SettingsGetStr(
		sNetId:='',
		hFile:=hSettingsFile,
		bExecute:=bSettingsGetStrExecute,
		tTimeout:=T#1S,
		bBusy=>bSettingsGetStrBusy,
		bError=>bSettingsGetStrError,
		nErrId=>nSettingsGetStrError,
		sLine=>sSettingsGetStr,
		bEOF=>bGetStrSettingsEOF
);
		
SettingsClose(
		sNetId:='',
		hFile:=hSettingsFile,
		bExecute:=bSettingsCloseExecute,
		tTimeout:=T#5S,
		bBusy=>bSettingsCloseBusy,
		bError=>bSettingsCloseError,
		nErrId=>nSettingsCloseError
		);

END_PROGRAM

// ---- POUs/GENERAL/Components/Robot/ROBOTREMOTE.TcPOU
PROGRAM ROBOTREMOTE
VAR_INPUT
	bRobotCommOpenEnable : BOOL := FALSE;
	bRobotCommCloseEnable: BOOL := FALSE;
	bRobotCommandSend : BOOL := FALSE;
	sRobotCommand : STRING := '';
	sRobotCommandParam1 : STRING := '';
	sRobotCommandParam2 : STRING := '';
	sRobotCommandParam3 : STRING := '';
	sRobotCommandParam4 : STRING := '';
	sRobotCommandParam5 : STRING := '';
END_VAR
VAR_OUTPUT
	bRobotCommOpen : BOOL := FALSE;
	nRobotErrId: UDINT;
	sRobotResult : STRING := '';
	iState: INT := 0;
END_VAR
VAR	
//LOCALS
	//RobotComm
	sRobotRemoteHost: STRING := '192.168.1.100';
//	sRobotRemoteHost: STRING := '192.168.1.22';
	bConnectBusy: BOOL;
	bSendBusy: BOOL;
	bReceiveBusy: BOOL;
	bCloseBusy: BOOL;
	bConnectError: BOOL;
	bSendError: BOOL;
	bReceiveError: BOOL;
	bCloseError: BOOL;
	nConnectErrId: UDINT;
	nSendErrId: UDINT;
	nReceiveErrId: UDINT;
	nCloseErrId: UDINT;
	hRobotSocket: T_HSOCKET;
	Delay: TON;
	bStartDelay: BOOL := FALSE;
	tDelay: TIME;
	rDelay: REAL;
	bDelayTimePassed: BOOL;
	
	//Kapcsolat nyitás
	bRobotSocketOpenEnable: BOOL := FALSE;
	RobotSocketOpen: FB_SocketConnect;
	iOpenTrials: INT;
	
	//Küldés
	bExecuting : BOOL := FALSE;
	bRobotSocketSendEnable: BOOL := FALSE;
	RobotSocketSend: FB_SocketSend;
	sLRobotCommandForResult: STRING :='';
	sLRobotCommand: STRING :='';
	sLRobotParam1: STRING :='';
	sLRobotParam2: STRING :='';
	sLRobotParam3: STRING :='';
	sLRobotParam4: STRING :='';
	sLRobotParam5: STRING :='';
	sRobotSendData: STRING;
	uSendByteLen: UDINT := 0;
	baSendByteArray: ARRAY[0..255] OF BYTE;
	bRobotSocketReceiveEnable: BOOL := FALSE;
	RobotSocketReceive: FB_SocketReceive;
	sRobotReceived: STRING :='';
	nRobotReceivedBytesNum: UDINT;
	baReceivedByteArray: ARRAY[0..255] OF BYTE;
	iTemp : INT := 0;
	
	//Fogadás kiértékelés
	fb_ResultSplitter : fb_SplitRobotResult;
	bIsError : BOOL;
	sErrorOrResult : STRING;
	
	//Kapcsolat bontás
	bRobotSocketCloseEnable: BOOL := FALSE;
	RobotSocketClose: FB_SocketClose;
	bRobotSocketbusy: BOOL;
END_VAR

rDelay:=TIME_TO_REAL(tDelay);

RobotSocketOpen(
			sSrvNetId:= '', 
			sRemoteHost:= sRobotRemoteHost, 
			nRemotePort:= 5000, 
			bExecute:= bRobotSocketOpenEnable, 
			tTimeout:= T#90S, 
			bBusy=> bConnectBusy, 
			bError=> bConnectError, 
			nErrId=> nConnectErrId, 
			hSocket=> hRobotSocket);
			
RobotSocketSend(
		sSrvNetId:= '', 
		hSocket:= hRobotSocket, 
		cbLen:= uSendByteLen, 
		pSrc:= ADR(baSendByteArray), 
		bExecute:= bRobotSocketSendEnable, 
		tTimeout:= T#5S, 
		bBusy=> bSendBusy, 
		bError=> bSendError, 
		nErrId=> nSendErrId);
		
RobotSocketReceive(
	sSrvNetId:= '', 
	hSocket:= hRobotSocket, 
	cbLen:= 255, 
	pDest:= ADR(baReceivedByteArray), 
	bExecute:= bRobotSocketReceiveEnable, 
	tTimeout:= T#5S, 
	bBusy=> bReceiveBusy, 
	bError=> bReceiveError, 
	nErrId=> nReceiveErrId, 
	nRecBytes=> nRobotReceivedBytesNum);		
		
RobotSocketClose(
	sSrvNetId:= '', 
	hSocket:= hRobotSocket, 
	bExecute:= bRobotSocketCloseEnable, 
	tTimeout:= T#90S, 
	bBusy=> bCloseBusy, 
	bError=> bCloseError, 
	nErrId=> nCloseErrId);

//Kommunikáció nyitás
IF (bRobotCommOpenEnable = TRUE) AND (bRobotCommOpen = FALSE) AND (iState <= 0) THEN
	iState:=1;
	iOpenTrials:=0;
	bIsError:=FALSE;
END_IF;

//Parancs küldés
IF (bRobotCommandSend = TRUE) AND (bRobotCommOpen=TRUE) AND(iState <= 0) THEN
	iState:=11;
	bIsError:=FALSE;
END_IF;
//Kommunikáció zárás
IF (bRobotCommCloseEnable = TRUE) AND (bRobotCommOpen = TRUE) AND (iState <= 0) THEN
	iState:=31;
	bIsError:=FALSE;
END_IF;




CASE iState OF
	
	1:	//Kommunikáció nyitás
		bRobotSocketOpenEnable:=TRUE;
		iState:=2;
	
	2:
		IF bConnectBusy = TRUE THEN
			iState:=3;
		END_IF
	3:
		IF bConnectBusy = FALSE THEN
			iState:=4;
		END_IF 
		
	4:
		IF bConnectError =FALSE THEN
			//Minden OK
			bRobotCommOpen:=TRUE;
			iState:=0;
		ELSE
			//HIBA
			iOpenTrials:=iOpenTrials+1;
			bRobotCommOpen:=FALSE;
			IF iOpenTrials<6 THEN
				bConnectError:=FALSE;
				iState:=5;
				bStartDelay:=TRUE;
				tDelay:=T#10S;
			ELSE
				iOpenTrials:=0;
				bStartDelay:=FALSE;
				iState:=0;
			END_IF
		END_IF
		bRobotCommOpenEnable := FALSE;
		bRobotSocketOpenEnable:=FALSE;
	5:
		IF bDelayTimePassed=TRUE THEN
			bStartDelay:=FALSE;
			iState:=1;
		END_IF
		
		
	11: //Parancs küldés
		nRobotErrId := 0;
		sLRobotCommandForResult := sRobotCommand;
		sLRobotCommand := sRobotCommand;
		sLRobotParam1 := sRobotCommandParam1;
		sLRobotParam2 := sRobotCommandParam2;
		sLRobotParam3 := sRobotCommandParam3;
		sLRobotParam4 := sRobotCommandParam4;
		sLRobotParam5 := sRobotCommandParam5;
		sRobotSendData := f_RobotCommandTranslation(sLRobotCommand,sLRobotParam1,sLRobotParam2,sLRobotParam3,sLRobotParam4,sLRobotParam5);
		baSendByteArray := MAXSTRING_TO_BYTEARR(sRobotSendData);
		uSendByteLen := INT_TO_UDINT(LEN(sRobotSendData));
		MEMSET(ADR(baReceivedByteArray), 0, 256);
		
		iState:=12;
		
	12:
		bRobotSocketSendEnable:=TRUE;
		iState:=13;
		
	13:
		IF bSendBusy = TRUE THEN
			iState:=14;
		END_IF
	14:
		IF bSendBusy = FALSE THEN
			iState:=15;
		END_IF 
		
	15:
		IF bSendError =FALSE THEN
			//Minden OK
			bIsError:= FALSE;
			iState:=21;
		ELSE
			//HIBA
			bIsError:= TRUE;	
			iState:=0;
		END_IF
		bRobotCommandSend := FALSE;
		bRobotSocketSendEnable:=FALSE;
		
		sRobotCommand:='';
		sRobotCommandParam1 := '';
		sRobotCommandParam2 := '';
		sRobotCommandParam3 := '';
		sRobotCommandParam4 := '';
		sRobotCommandParam5 := '';
		
		sLRobotCommand := '';
		sLRobotParam1 := '';
		sLRobotParam2 := '';
		sLRobotParam3 := '';
		sLRobotParam4 := '';
		sLRobotParam5 := '';
		
	21:	//Adatfogadás
		nRobotReceivedBytesNum:=0;
		bRobotSocketReceiveEnable := TRUE;
		iState:=22;
		
	22:
		IF bReceiveBusy = TRUE THEN
			iState:=23;
		END_IF
	23:
		IF bReceiveBusy = FALSE THEN
			iState:=24;
		END_IF 
		
	24:
		IF bReceiveError =FALSE THEN
			//Minden OK
			bIsError:= FALSE;
			iState:=25;
		ELSE
			//HIBA
			bIsError:= TRUE;
			iState:=0;	
		END_IF
		bRobotSocketReceiveEnable:=FALSE;
		
	25:
		IF (nRobotReceivedBytesNum <>0) THEN
			sRobotReceived := BYTEARR_TO_MAXSTRING(baReceivedByteArray);
			fb_ResultSplitter(sCommand:= sLRobotCommandForResult, sResult:= sRobotReceived, bIsError=> bIsError, sErrorOrResult=> sErrorOrResult);
			IF bIsError THEN
				nRobotErrId:=STRING_TO_UDINT(sErrorOrResult);
				sRobotResult:='';
			ELSE
				nRobotErrId:=0;
				sRobotResult:=sErrorOrResult;
			END_IF
			iState:=0;
		ELSE
			iState:=21;
		END_IF
		
	31:	//Kommunikáció zárás
		bRobotSocketCloseEnable:=TRUE;
		iState:=32;
	
	32:
		IF bCloseBusy = TRUE THEN
			iState:=33;
		END_IF
	33:
		IF bCloseBusy = FALSE THEN
			iState:=34;
		END_IF 
		
	34:
		IF bCloseError =FALSE THEN
			//Minden OK
			bRobotCommOpen:=FALSE;
		ELSE
			//HIBA
			bRobotCommOpen:=FALSE;	//még át kell gondolni
		END_IF
		bRobotCommCloseEnable := FALSE;
		bRobotSocketCloseEnable:=FALSE;
		iState:=0;
	
END_CASE
Delay(IN:=bStartDelay, PT:=tDelay, Q=>bDelayTimePassed, ET=>);

END_PROGRAM

// ---- POUs/GENERAL/Helpers/fb_SplitRobotResult.TcPOU
FUNCTION_BLOCK fb_SplitRobotResult
VAR_INPUT
	sCommand : STRING;
	sResult : STRING;
END_VAR
VAR_OUTPUT
	bIsError : BOOL;
	sErrorOrResult : STRING;
END_VAR
VAR
	sCRLFString : STRING := '  ';
	nCRLFPosition : INT := 0;
	sTempResult : STRING;
END_VAR

sCRLFString[0] := 16#D;
sCRLFString[1] := 16#A;
IF MID(sResult,LEN(sCommand),2)=sCommand THEN
	sErrorOrResult := MID(sResult,LEN(sResult)-LEN(sCommand)-4,3+LEN(sCommand));
	nCRLFPosition := FIND(sErrorOrResult,sCRLFString);
	IF nCRLFPosition > 0 THEN
		sErrorOrResult := DELETE(sErrorOrResult,2,nCRLFPosition);
	END_IF
	IF sResult[0] = 16#23 THEN
		bIsError := FALSE;
	ELSE
		bIsError := TRUE;
	END_IF
ELSE
	bIsError := TRUE;
	sErrorOrResult := '1';
END_IF

END_FUNCTION_BLOCK

// ---- POUs/GENERAL/Helpers/f_RobotCommandTranslation.TcPOU
FUNCTION f_RobotCommandTranslation : STRING
VAR_INPUT
	sCommand : STRING;
	sParam1 : STRING;
	sParam2 : STRING;
	sParam3 : STRING;
	sParam4 : STRING;
	sParam5 : STRING;
END_VAR
VAR
	uLength : INT := 0;
	tempTranslation : STRING := '';
	nDollarPosition : INT := 0;
	sDollarString : STRING := ' ';
END_VAR

//IF sCommand='Login' THEN
//	f_RobotCommandTranslation := CONCAT(' Login,',sParam1);
//END_IF
//IF sCommand='LOGOUT' THEN
//	f_RobotCommandTranslation:=' Logout';
//END_IF
//Kezdő $ karakter
sDollarString[0] := 16#24;
tempTranslation := CONCAT(' ',sCommand);
tempTranslation[0] := 16#24;

//Ha van Paraméter1 akkor berakjuk
IF sParam1<>'' THEN
	tempTranslation := CONCAT(tempTranslation,',');
	tempTranslation := CONCAT(tempTranslation,sParam1);
END_IF

//Ha van Paraméter2 akkor berakjuk
IF sParam2<>'' THEN
	tempTranslation := CONCAT(tempTranslation,',');
	tempTranslation := CONCAT(tempTranslation,sParam2);
END_IF

//Ha van Paraméter3 akkor berakjuk
IF sParam3<>'' THEN
	tempTranslation := CONCAT(tempTranslation,',');
	tempTranslation := CONCAT(tempTranslation,sParam3);
END_IF

//Ha van Paraméter4 akkor berakjuk
IF sParam4<>'' THEN
	tempTranslation := CONCAT(tempTranslation,',');
	tempTranslation := CONCAT(tempTranslation,sParam4);
END_IF

//Ha van Paraméter5 akkor berakjuk
IF sParam5<>'' THEN
	tempTranslation := CONCAT(tempTranslation,',');
	tempTranslation := CONCAT(tempTranslation,sParam5);
END_IF

//Add CRLF to end
tempTranslation := CONCAT(tempTranslation,'  ');
tempTranslation[LEN(tempTranslation)-2]:=16#D;
tempTranslation[LEN(tempTranslation)-1]:=16#A;
nDollarPosition := FIND(tempTranslation,'dollar');
IF nDollarPosition > 0 THEN
	tempTranslation := DELETE(tempTranslation,6,nDollarPosition);
	tempTranslation := INSERT(tempTranslation,sDollarString,nDollarPosition-1);
END_IF
f_RobotCommandTranslation:=tempTranslation;

END_FUNCTION

// ---- POUs/PISTI/Components/Laser.TcPOU
PROGRAM Laser
VAR_INPUT
	s_InCommand : STRING :='';
	s_TypeCode : STRING :='0';	
END_VAR
VAR_OUTPUT
	s_Result: STRING;
END_VAR
VAR
	iState: INT;
	iState2: INT;
	iTrials: INT;
	iSetPower: INT;
	iWishPower: INT := 12;
	sWishPower: STRING;
	sSetPower: STRING;

	// Laser Com Open
	sLaserRemoteHost: STRING := '192.168.1.99';
//	sLaserRemoteHost: STRING := '192.168.1.22';
	LaserSocketOpen: FB_SocketConnect;
	bLaserSocketOpenEnable: BOOL := FALSE;
	bLaserSocketBusy: BOOL;
	bLaserSocketError: BOOL;
	nLaserSocketErrId: UDINT;
	hLaserSocket: T_HSOCKET;
	
	// Laser Send
	LaserSocketSend: FB_SocketSend;
	uSendByteLen: UDINT := 0;
	baSendByteArray: ARRAY[0..255] OF BYTE;
	bLaserSocketSendEnable: BOOL := FALSE;
	bLaserSendbusy: BOOL;
	bLaserSendError: BOOL;
	nLaserSendErrId: UDINT;

	// Laser Receive
	LaserSocketReceive: FB_SocketReceive;
	baReceivedByteArray: ARRAY[0..255] OF BYTE;
	bLaserSocketReceiveEnable: BOOL := FALSE;
	bLaserReceiveBusy: BOOL;
	bLaserReceiveError: BOOL;
	nLaserReceiveErrId: UDINT;
	nLaserReceivedBytesNum: UDINT;
	
	// Laser Com Close
	LaserSocketClose: FB_SocketClose;
	bLaserSocketCloseEnable: BOOL := FALSE;
	bLaserSocketCloseBusy: BOOL;
	bLaserSocketCloseError: BOOL;
	nLaserSocketCloseErrId: UDINT;
	
	sLaserSend: STRING :='';
	sLaserReceived: STRING :='';
	sExpectedResponse: STRING := '';
	
	// Lézer szoftver megnyitása
	FB_Start_FOBA_Draw: NT_StartProcess;
	bStartFOBADraw: BOOL;
	bFOBADrawBusy: BOOL;
	bFOBADrawErr: BOOL;
	nFOBADrawErr: UDINT;

	// Lézer parancs lista megnyitása
	FB_Start_Ultimate: NT_StartProcess;
	bStartUltimate: BOOL;
	bUltimateBusy: BOOL;
	bUltimateErr: BOOL;
	nUltimateErr: UDINT;
	
END_VAR

CASE iState OF
	0:	// Parancsértelmezés
		iState:=1;
		iTrials:=0;
		sExpectedResponse:='$06;0000;$R$N';
		IF s_InCommand='GETJOB' THEN
			sLaserSend:='GetJob;';
		ELSIF s_InCommand='SETJOB_637' THEN
			sLaserSend:='SetJob;637xxx;';
		ELSIF s_InCommand='SETJOB_745900' THEN
			sLaserSend:='SetJob;745900;';
		ELSIF s_InCommand='SETJOB_745910' THEN
			sLaserSend:='SetJob;745910;';
		ELSIF s_InCommand='SETJOB_521' THEN
			sLaserSend:='SetJob;521950;';
		ELSIF s_InCommand='START' THEN
			sLaserSend:='Start;';
		ELSIF (s_InCommand='SETTYPE') THEN
			IF (GVL.iSelectedProductType<8) THEN // 637 esetén
				s_TypeCode:=TO_STRING(GVL.iSelectedProductType);
			ELSIF (GVL.iSelectedProductType>8) THEN // 745 esetén
				CASE GVL.iSelectedProductType OF
					9, 10: s_TypeCode:='0'; //745900 és 745910
					11, 12: s_TypeCode:='1'; //745905 és 745915
					13, 14: s_TypeCode:='2'; //745906 és 745916
					15, 16: s_TypeCode:='3'; //745907 és 745917
				END_CASE
			END_IF;
			sLaserSend:=CONCAT('SetVars;TypeCode;',CONCAT(s_TypeCode,';'));
		ELSIF s_InCommand='GETSTATUS' THEN
			sLaserSend:='GetStatus;';
			s_Result:='';
		ELSIF s_InCommand='GETINTENSITY' THEN
			sLaserSend:='GetIntensity;';
			s_Result:='';
		ELSE
			iState:=0;
		END_IF			
	1:	// Vár arra, hogy ne legyen folyamatban a socket megnyitása
		IF (bLaserSocketBusy=FALSE) THEN
			iState:=2;
		END_IF							
	2:	// Ha nincs nyitva a lézer socket, kezdeményezi a megnyitását
		IF NOT(GVL.bLaserCommOpen) THEN
			bLaserSocketOpenEnable:=TRUE;
			IF (bLaserSocketBusy=TRUE) THEN
				iState:=3;
			END_IF				
		ELSE
			iState:=4;
		END_IF
	3:	// Vár, hogy megnyíljon a lézer socket
		IF (bLaserSocketBusy=FALSE) AND (bLaserSocketError=FALSE) THEN
			GVL.bLaserCommOpen:=TRUE;
			bLaserSocketOpenEnable:=FALSE;
			iState:=4;
		ELSIF (bLaserSocketError=TRUE) THEN
			GVL.bLaserCommOpen:=FALSE;
			bLaserSocketOpenEnable:=FALSE;
			iState:=2;
		END_IF
	4:	// Ha nincs folyamatban parancsküldés, kezdeményezi a parancsküldést
		IF (bLaserSendBusy=FALSE) THEN
			MEMSET(ADR(baSendByteArray), 0, 256); // Byte tömb ürítése
			baSendByteArray := MAXSTRING_TO_BYTEARR(sLaserSend); // Parancs string byte tömbbe
			uSendByteLen := INT_TO_UDINT(LEN(sLaserSend)); // Parancs string hossza
			baSendByteArray[uSendByteLen]:=16#D; // Lezáró karakter 1
			baSendByteArray[uSendByteLen+1]:=16#A; // Lezáró karakter 2
			bLaserSocketSendEnable:=TRUE; // Küldés indítójel
			iState:=5;
		END_IF
	5:	// Vár, hogy a parancsküldés elkezdődjön
		IF (bLaserSendBusy=TRUE) THEN
			iState:=6;
		END_IF
	6:	// Vár a parancsküldés sikeres befejezésére
		IF (bLaserSendBusy=FALSE) AND (bLaserSendError=FALSE) THEN
			bLaserSocketSendEnable:=FALSE;
			iState:=7;
		END_IF
	7:	// Ha nincs folyamatban válaszfogadás, kezdeményezi a válaszfogadást
		IF (bLaserReceiveBusy=FALSE) THEN
			MEMSET(ADR(baReceivedByteArray), 0, 256); // Byte tömb ürítése
			bLaserSocketReceiveEnable:=TRUE; // Fogadás indítójel
			iState:=8;
		END_IF
	8:	// Vár, hogy a válaszfogadás elkezdődjön
		IF (bLaserReceiveBusy=TRUE) THEN
			iState:=9;
		END_IF
	9:	// Vár a válaszfogadás sikeres befejezésére
		IF (bLaserReceiveBusy=FALSE) AND (bLaserReceiveError=FALSE) THEN
			bLaserSocketReceiveEnable:=FALSE;
			sLaserReceived := BYTEARR_TO_MAXSTRING(baReceivedByteArray);
			MEMSET(ADR(baReceivedByteArray), 0, 256);
			iState:=10;
		END_IF
	10:	// Kiértékelés
		IF (sLaserReceived=sExpectedResponse) THEN
			s_InCommand:='';
		ELSE
			IF iTrials<5 THEN
				iTrials:=iTrials+1;
				iState:=7;
			ELSE
				s_InCommand:=sLaserReceived;
			END_IF
		END_IF
		sExpectedResponse:='';
		iState:=0;
		IF sLaserSend='GetStatus;' THEN
			IF (FIND(sLaserReceived,'LaserStatusReady')>0)
				OR (FIND(sLaserReceived,'LaserStatusStandby')>0) THEN
				s_Result:='READY';
			ELSE
				s_Result:='NOT_READY';
			END_IF
		ELSIF LEFT(sLaserSend,12)='GetIntensity' THEN
			sSetPower:=DELETE(sLaserReceived,8,0);
			sSetPower:=LEFT(sSetPower,LEN(sSetPower)-3);
			iSetPower:=STRING_TO_INT(sSetPower);
//			sLaserSend:='GetIntensity;';
			;
		ELSIF LEFT(sLaserSend,12)='SetIntensity' THEN
			sLaserSend:='GetIntensity;';
			iState:=1;
		END_IF
END_CASE

// FOBA Draw indítási állapotgép
CASE iState2 OF
	0:	// Várakozás parancsra
		IF (bStartFOBADraw=TRUE) THEN
			iState2:=1;
		ELSIF (bStartUltimate=TRUE) THEN
			iState2:=11;
		END_IF
	1:
		IF (bFOBADrawBusy=TRUE) THEN
			iState2:=2;
		END_IF
	2:
		IF (bFOBADrawBusy=FALSE) THEN
			bStartFOBADraw:=FALSE;
			iState2:=0;
		END_IF
	11:
		IF (bUltimateBusy=TRUE) THEN
			iState2:=12;
		END_IF
	12:
		IF (bUltimateBusy=FALSE) THEN
			bStartUltimate:=FALSE;
			iState2:=0;
		END_IF
END_CASE

// Kommunikáció nyitás
LaserSocketOpen(
	sSrvNetId:= '', 
	sRemoteHost:= sLaserRemoteHost, 
	nRemotePort:= 20001, 
	bExecute:= bLaserSocketOpenEnable, 
	tTimeout:= T#45S, 
	bBusy=> bLaserSocketBusy, 
	bError=> bLaserSocketError, 
	nErrId=> nLaserSocketErrId, 
	hSocket=> hLaserSocket);

// Parancsküldés
LaserSocketSend(
	sSrvNetId:= '', 
	hSocket:= hLaserSocket, 
	cbLen:= uSendByteLen + 2, 
	pSrc:= ADR(baSendByteArray), 
	bExecute:= bLaserSocketSendEnable, 
	tTimeout:= T#5S, 
	bBusy=> bLaserSendBusy,
	bError=> bLaserSendError,
	nErrId=> nLaserSendErrId);

// Válasz fogadása
LaserSocketReceive(
	sSrvNetId:= '', 
	hSocket:= hLaserSocket, 
	cbLen:= 255, 
	pDest:= ADR(baReceivedByteArray), 
	bExecute:= bLaserSocketReceiveEnable, 
	tTimeout:= T#5S, 
	bBusy=> bLaserReceiveBusy, 
	bError=> bLaserReceiveError, 
	nErrId=> nLaserReceiveErrId, 
	nRecBytes=> nLaserReceivedBytesNum
);

//Kommunikáció bontás
LaserSocketClose(
	sSrvNetId:= '', 
	hSocket:= hLaserSocket, 
	bExecute:= bLaserSocketCloseEnable, 
	tTimeout:= T#45S, 
	bBusy=> bLaserSocketCloseBusy, 
	bError=> bLaserSocketCloseError, 
	nErrId=> nLaserSocketCloseErrId);

// Lézer saját szoftverének indítása
FB_Start_FOBA_Draw(
					NETID:='',
					PATHSTR:='C:\Program Files\FOBA\FOBA Draw\FOBA Draw 9.2.2\FOBA Draw.exe',
					DIRNAME:='C:\Program Files\FOBA\FOBA Draw\FOBA Draw 9.2.2\',
					COMNDLINE:='',
					START:=bStartFOBADraw,
					TMOUT:=T#30S,
					BUSY => bFOBADrawBusy,
					ERR => bFOBADrawErr,
					ERRID => nFOBADrawErr
					);

// Lézer parancs listájának megnyitása
FB_Start_Ultimate(
					NETID:='',
					PATHSTR:='C:\Program Files\Adobe\Reader 11.0\Reader\AcroRd32.exe',
					DIRNAME:='C:\637\',
					COMNDLINE:='"C:\637\Specification_Ultimate_V1.5.1_Foba_Rev2.pdf"',
					START:=bStartUltimate,
					TMOUT:=T#30S,
					BUSY => bUltimateBusy,
					ERR => bUltimateErr,
					ERRID => nUltimateErr
					);

END_PROGRAM

// ---- POUs/JOZSI/Components/NTC.TcPOU
PROGRAM NTC
VAR_INPUT
	bVagashoz : BOOL := FALSE;

	//Gombok funkcióváltása
	bVagasGombbal : BOOL;
	bVagoFelLeGombbal : BOOL;
END_VAR
VAR
	
	//IO
	bZoldGomb AT %I*: BOOL;
	bPirosGomb AT %I*: BOOL;
	bNTCLaberzekeloBal AT %I*: BOOL;
	bNTCLaberzekeloJobb AT %I*: BOOL;
	bNTCFekBal AT %Q*: BOOL := FALSE;
	bNTCFekJobb AT %Q*: BOOL := FALSE;
	
	
	//MOTOR
	bZeroSpeed AT %I*: BOOL;
	bSpeedReached AT %I*: BOOL;
	bReady AT %I*: BOOL;
	bAlarm AT %I*: BOOL;
	bServoON AT %Q*: BOOL := TRUE;
	bReverseRotationStart AT %Q*: BOOL := FALSE;
	bForwardRotationStart AT %Q*: BOOL := FALSE;
	bSpeed1 AT %Q*: BOOL := TRUE;
	bReset AT %Q*: BOOL := FALSE;
	
	//VARS
	bInternalState : BOOL := FALSE;
	iDelayFor : INT := 0;
	iTemp : INT := 0;
	bJogPlus : BOOL := FALSE;
	bJogMinus : BOOL := FALSE;
	bElozoLab : BOOL := FALSE;
	
	
END_VAR

IF (bVagasGombbal=FALSE) AND (bVagoFelLeGombbal=FALSE) THEN
	IF ((bZoldGomb=TRUE OR bJogPlus=TRUE) AND bAlarm=TRUE AND bServoON=TRUE AND bReady=TRUE) THEN
		bForwardRotationStart := TRUE;
		bReverseRotationStart := FALSE;
		bVagashoz:=FALSE;
		bInternalState:=FALSE;
	ELSE
		IF bInternalState=FALSE THEN
			bForwardRotationStart := FALSE;
		END_IF
	END_IF
	IF ((bPirosGomb=TRUE OR bJogMinus=TRUE) AND bAlarm=TRUE AND bServoON=TRUE AND bReady=TRUE) THEN
		bReverseRotationStart := TRUE;
		bForwardRotationStart := FALSE;
		bVagashoz:=FALSE;
		bInternalState:=FALSE;
	ELSE
		IF bInternalState=FALSE THEN
			bReverseRotationStart := FALSE;
		END_IF
	END_IF
ELSIF (bVagoFelLeGombbal=TRUE) AND (NTCProcess.s_InCommand='')
		AND ((bZoldGomb=TRUE) OR (bPirosGomb=TRUE)) THEN
	NTCProcess.s_InCommand:='VAGO_FEL-LE';
ELSIF (bZoldGomb=TRUE) AND (NTCProcess.s_InCommand='') THEN
	NTCProcess.s_InCommand:='VAGAS';
ELSIF (bPirosGomb=TRUE) AND (NTCProcess.s_InCommand='') THEN
	NTCProcess.s_InCommand:='NTC_ELENGED';
END_IF;

(*// Új NTC pozícionáló algoritmus (két lábérzékelő + két fék)	
IF (bVagashoz=TRUE AND bAlarm=TRUE AND bServoON=TRUE AND bReady=TRUE) THEN
	bInternalState := TRUE;
	bVagashoz:=FALSE;
	IF (bNTCLaberzekeloBal=TRUE) AND (bNTCLaberzekeloJobb=TRUE) THEN
		bElozoLab := TRUE;
	END_IF
END_IF
		
IF bInternalState=TRUE THEN
//	IF (bNTCLaberzekeloBal=TRUE) AND (bNTCLaberzekeloJobb=TRUE) THEN		
	IF (bNTCFekBal=TRUE) AND (bNTCFekJobb=TRUE) THEN		
		bNTCFekBal:=FALSE;
		bNTCFekJobb:=FALSE;
		IF bElozoLab=FALSE THEN
			bForwardRotationStart := FALSE;
			bInternalState := FALSE;
		ELSE
			bForwardRotationStart := TRUE;
		END_IF
	ELSIF (bNTCLaberzekeloBal=TRUE) THEN
		bNTCFekBal:=TRUE;
	ELSIF (bNTCLaberzekeloJobb=TRUE) THEN
		bNTCFekJobb:=TRUE;
	ELSE	
		IF bElozoLab = TRUE THEN
			bElozoLab := FALSE;
		END_IF;
		bForwardRotationStart := TRUE;
	END_IF
END_IF
*)
// Régi NTC pozícionáló algoritmus: csak egy lábérzékelő fékek nélkül
IF (bVagashoz=TRUE AND bAlarm=TRUE AND bServoON=TRUE AND bReady=TRUE) THEN
	bInternalState := TRUE;
	bVagashoz:=FALSE;
	IF(bNTCLaberzekeloJobb=TRUE) THEN
		bElozoLab := TRUE;
	END_IF
END_IF
		
IF bInternalState=TRUE THEN
	IF(bNTCLaberzekeloJobb=TRUE) THEN
		IF bElozoLab=FALSE THEN
			bForwardRotationStart := FALSE;
			bInternalState := FALSE;
		ELSE
			bForwardRotationStart := TRUE;
		END_IF
	ELSE
		IF bElozoLab = TRUE THEN
			bElozoLab := FALSE;
		END_IF;
		bForwardRotationStart := TRUE;
	END_IF
END_IF

END_PROGRAM

// ---- POUs/JOZSI/Components/NTCProcess.TcPOU
PROGRAM NTCProcess
VAR_INPUT
	s_InCommand : STRING := '';
	s_InCommandParam1 : STRING := '';
	s_InCommandParam2 : STRING := '';
	s_InCommandParam3 : STRING := '';
	s_InCommandParam4 : STRING := '';
	s_InCommandParam5 : STRING := '';
END_VAR
VAR_OUTPUT
	n_OutErrId: UINT;
END_VAR
VAR
	//IO
	bVagoHajlitoFent AT %I*: BOOL;
	bVagoHajlitoLent AT %I*: BOOL;
	bKiszedoKint AT %I*: BOOL;
	bKiszedoBent AT %I*: BOOL;
	bMegfogoNyitva AT %I*: BOOL;
	bMegfogoZarva AT %I*: BOOL;
	bVagoHajlito AT %Q*: BOOL := FALSE;
	bKiszedo AT %Q*: BOOL := FALSE;
	bMegfogo AT %Q*: BOOL := FALSE;
	
	//INTERNAL	
	iState : INT := 0;
	s_InLCommand : STRING := '';
	T_Ticker : TON;
	bTickerEnable : BOOL := FALSE;
	tTickerTime : TIME := T#3000MS;
	bTickerQ : BOOL := FALSE;
END_VAR

IF NTCProcess.s_InCommand <>'' AND s_InLCommand = '' THEN
	s_InLCommand := NTCProcess.s_InCommand;
END_IF
IF s_InLCommand <> '' THEN
//	IF iState = 0 AND s_InLCommand = 'VAGAS' THEN
//		iState := 1;
//	END_IF
	IF iState = 0 THEN 
		IF s_InLCommand = 'VAGAS' THEN
			iState := 1;
		ELSIF s_InLCommand = 'NTC_ELENGED' THEN
			iState := 21;
		ELSIF s_InLCommand = 'VAGO_FEL-LE' THEN
			iState := 31;
		END_IF
	END_IF
	CASE iState OF 
		1:
			IF (bVagoHajlitoFent = TRUE AND bVagoHajlitoLent = FALSE
				AND bKiszedoBent = FALSE AND bKiszedoKint = TRUE
				AND bMegfogoZarva = FALSE AND bMegfogoNyitva = TRUE
				AND NTC.bInternalState=FALSE) THEN
				n_OutErrId := 0;
				iState := 2;
			ELSE
				IF MAIN.bLevegoOK = FALSE THEN
					n_OutErrId := 5;
				ELSIF bVagoHajlitoFent = FALSE THEN
					n_OutErrId := 115;
				ELSIF bVagoHajlitoLent = TRUE THEN
					n_OutErrId := 114;
				ELSIF bKiszedoBent = TRUE THEN
					n_OutErrId := 136;
				ELSIF bKiszedoKint = FALSE THEN
					n_OutErrId := 133;
				ELSIF bMegfogoZarva = TRUE THEN 
					n_OutErrId := 132;
				ELSIF bMegfogoNyitva = FALSE THEN
					n_OutErrId := 129;
				ELSIF NTC.bInternalState=TRUE THEN
					n_OutErrId := 300;
				END_IF;
				iState := 0;
			END_IF
		2:
			NTC.bVagashoz := TRUE;
			iState := 3;
		3:
			IF (NTC.bInternalState = FALSE AND NTC.bVagashoz = FALSE) THEN
				iState := 4;
				n_OutErrId := 0;
			ELSIF NTC.bInternalState=TRUE THEN
				n_OutErrId := 300;
			ELSIF NTC.bVagashoz = TRUE THEN
				n_OutErrId := 301;
			END_IF
		4:
			bKiszedo := TRUE;
			iState := 5;
		5:
			IF bKiszedoBent = TRUE AND bKiszedoKint = FALSE THEN
				n_OutErrId := 0;
				tTickerTime:=T#1S;
				bTickerEnable := FALSE;
				iState := 6;
			ELSIF MAIN.bLevegoOK = FALSE THEN
				n_OutErrId := 5;
			ELSIF bKiszedoBent = FALSE THEN
				n_OutErrId := 135;
			ELSIF bKiszedoKint = TRUE THEN
				n_OutErrId := 134;
			END_IF
		6:
			bTickerEnable := TRUE;
			iState := 7;
		7:
			IF bTickerQ = TRUE THEN
				bTickerEnable := FALSE;
				iState := 8;
			END_IF
		8:
			bVagoHajlito := TRUE;
			iState := 9;
		9:
			IF bVagoHajlitoLent = TRUE AND bVagoHajlitoFent = FALSE THEN
				n_OutErrId := 0;
				tTickerTime:=T#1S;
				bTickerEnable := FALSE;
				iState := 10;
			ELSIF MAIN.bLevegoOK = FALSE THEN
				n_OutErrId := 5;
			ELSIF bVagoHajlitoLent = FALSE THEN 
				n_OutErrId := 113;
			ELSIF bVagoHajlitoFent = TRUE THEN
				n_OutErrId := 116;
			END_IF
		10:
			bTickerEnable := TRUE;
			iState := 11;
		11:
			IF bTickerQ = TRUE THEN
				bTickerEnable := FALSE;
				iState := 12;
			END_IF
		12:
			bVagoHajlito := FALSE;
			iState := 13;
		13:
			IF bVagoHajlitoLent = FALSE AND bVagoHajlitoFent = TRUE THEN
				n_OutErrId := 0;
				tTickerTime:=T#3S;
				bTickerEnable := FALSE;
				iState := 14;
			ELSIF MAIN.bLevegoOK = FALSE THEN
				n_OutErrId := 5;
			ELSIF bVagoHajlitoLent = TRUE THEN 
				n_OutErrId := 114;
			ELSIF bVagoHajlitoFent = FALSE THEN
				n_OutErrId := 115;
			END_IF
		14:
			bTickerEnable := TRUE;
			iState := 15;
		15:
			IF bTickerQ = TRUE THEN
				bTickerEnable := FALSE;
				iState := 16;
			END_IF
		16:
			bMegfogo := TRUE;
			iState := 17;
		17:
			IF bMegfogoZarva = TRUE AND bMegfogoNyitva = FALSE THEN
				n_OutErrId := 0;
				iState := 18;
			ELSIF MAIN.bLevegoOK = FALSE THEN
				n_OutErrId := 5;
			ELSIF bMegfogoZarva = FALSE THEN 
				n_OutErrId := 131;
			ELSIF bMegfogoNyitva = TRUE THEN
				n_OutErrId := 130;
			END_IF
		18:
			bKiszedo := FALSE;
			iState := 19;
		19:
			IF bKiszedoKint = TRUE AND bKiszedoBent = FALSE THEN
				n_OutErrId := 0;
				iState := 20;
			ELSIF MAIN.bLevegoOK = FALSE THEN
				n_OutErrId := 5;
			ELSIF bKiszedoKint = FALSE THEN 
				n_OutErrId := 133;
			ELSIF bKiszedoBent = TRUE THEN
				n_OutErrId := 136;
			END_IF
		20:
			iState := 0;
			n_OutErrId := 0;
		21:
			bMegfogo := FALSE;
			iState := 22;

		22:
			IF bMegfogoZarva = FALSE AND bMegfogoNyitva = TRUE THEN
				n_OutErrId := 0;
				iState := 20;
			ELSIF MAIN.bLevegoOK = FALSE THEN
				n_OutErrId := 5;
			ELSIF bMegfogoZarva = TRUE THEN 
				n_OutErrId := 132;
			ELSIF bMegfogoNyitva = FALSE THEN
				n_OutErrId := 129;
			END_IF

		31:
			IF (bVagoHajlitoFent = TRUE AND bVagoHajlitoLent = FALSE
				AND bKiszedoBent = FALSE AND bKiszedoKint = TRUE
				AND bMegfogoZarva = FALSE AND bMegfogoNyitva = TRUE
				AND NTC.bInternalState=FALSE) THEN
				n_OutErrId := 0;
				iState := 32;
			ELSE
				IF MAIN.bLevegoOK = FALSE THEN
					n_OutErrId := 5;
				ELSIF bVagoHajlitoFent = FALSE THEN
					n_OutErrId := 115;
				ELSIF bVagoHajlitoLent = TRUE THEN
					n_OutErrId := 114;
				ELSIF bKiszedoBent = TRUE THEN
					n_OutErrId := 136;
				ELSIF bKiszedoKint = FALSE THEN
					n_OutErrId := 133;
				ELSIF bMegfogoZarva = TRUE THEN 
					n_OutErrId := 132;
				ELSIF bMegfogoNyitva = FALSE THEN
					n_OutErrId := 129;
				ELSIF NTC.bInternalState=TRUE THEN
					n_OutErrId := 300;
				END_IF;
				iState := 0;
			END_IF
		32:
			bVagoHajlito := TRUE;
			iState := 33;
		33:
			IF bVagoHajlitoLent = TRUE AND bVagoHajlitoFent = FALSE THEN
				n_OutErrId := 0;
				tTickerTime:=T#1S;
				bTickerEnable := FALSE;
				iState := 34;
			ELSIF MAIN.bLevegoOK = FALSE THEN
				n_OutErrId := 5;
			ELSIF bVagoHajlitoLent = FALSE THEN 
				n_OutErrId := 113;
			ELSIF bVagoHajlitoFent = TRUE THEN
				n_OutErrId := 116;
			END_IF
		34:
			bTickerEnable := TRUE;
			iState := 35;
		35:
			IF bTickerQ = TRUE THEN
				bTickerEnable := FALSE;
				iState := 36;
			END_IF
		36:
			bVagoHajlito := FALSE;
			iState := 37;
		37:
			IF bVagoHajlitoLent = FALSE AND bVagoHajlitoFent = TRUE THEN
				n_OutErrId := 0;
				iState := 0;
			ELSIF MAIN.bLevegoOK = FALSE THEN
				n_OutErrId := 5;
			ELSIF bVagoHajlitoLent = TRUE THEN 
				n_OutErrId := 114;
			ELSIF bVagoHajlitoFent = FALSE THEN
				n_OutErrId := 115;
			END_IF

	END_CASE
	IF iState = 0 THEN
		NTCProcess.s_InCommand := '';
		s_InLCommand := '';
	END_IF
END_IF
T_Ticker(IN:= bTickerEnable, PT:= tTickerTime, Q=> bTickerQ, ET=> );

END_PROGRAM

// ---- POUs/GENERAL/Components/INIT.TcPOU
PROGRAM INIT
VAR
	iState: INT := -4;
	iStateHegeszto: INT := 0;		// Max 3
	iStateTCP: INT := 0;			// Max 5
	iStateLezer: INT := 0;			// Max 4
	iStateRobot: INT := 0;			// Max 8
	iStateHegesztoFejek: INT := 0;	// Max 3
	iStateVegmero: INT := 0;		// Max 3
	iStateNTCTengely: INT := 0;		// Max 5
	iStatePt1000Tengely: INT := 0;	// Max 5
	iStateHimba: INT := 0;			// Max 3
	bHegesztoKesz: BOOL := FALSE;
	bTCPKesz: BOOL := FALSE;
	bLezerKesz: BOOL := FALSE;
	bRobotKesz: BOOL := FALSE;
	bHegesztoFejekKesz: BOOL := FALSE;
	bVegmeroKesz: BOOL := FALSE;
	bNTCTengelyKesz: BOOL := FALSE;
	bPt1000TengelyKesz: BOOL := FALSE;
	bHimbaKesz: BOOL := FALSE;
	iKeszenletFoka: INT;
	CloseAllSocket: fb_SocketCloseAll;
	bExecuteCloseAll: BOOL;
	bCloseAllBusy: BOOL;
	bCloseAllError: BOOL;
	nCloseAllError: UDINT;
	TDelay: TON;
	
	// Indítási opciók
	bLevego: BOOL := TRUE;
	bRobot: BOOL := TRUE;
	bVegmero: BOOL := TRUE;
	bNTCTengely: BOOL := TRUE;
	bPt1000Tengely: BOOL := TRUE;
	bHegeszto: BOOL := TRUE;

	// Visualization indítása
	FB_Start_Visu: NT_StartProcess;
	bStartVisu: BOOL;
	bVisuBusy: BOOL;
	bVisuErr: BOOL;
	nVisuErr: UDINT;

	// Idő lekérdezése
	GetTime: NT_GetTime;
	bStartGetTime: BOOL;
	bGetTimeBusy: BOOL;
	bGetTimeError: BOOL;
	nGetTimeError: UDINT;
	tstDateTime: TIMESTRUCT;
	dtDateTime: DT;
	sYear: STRING;
	iState2: INT := 1;
	sMonth: STRING;
	sDay: STRING;
	sHour: STRING;
	sMinute: STRING;
	sSecond: STRING;

	WAIT: TON;
	bStartWait: BOOL := FALSE;
	bIdoLejart: BOOL := FALSE;
	
	FB_ShutDown: NT_Shutdown;	
	bStartShutDown: BOOL := FALSE;
	
	FB_RestartSystem: TC_Restart;
	bRestart: BOOL;
	bRestartBusy: BOOL;
	bRestartErr: BOOL;
	nRestartErr: UDINT;
	
	bStartDelay: BOOL;
	bDelayEnd: BOOL;
	// Max 5
	iStateKamera: INT;
	bKameraKesz: BOOL;
END_VAR

CASE iState OF
	-4:	// 1 ciklusnyi várakozás
		iState:=1;
	-3:	// Visu indító trigger
		bStartVisu:=TRUE;
		iState:=-2;
	-2:	// Várakozás az indító folyamat indulására
		IF (bVisuBusy=TRUE) THEN
			iState:=-1;
		END_IF
	-1:	// Várakozás a Visu indító folyamat befejeztére
		IF (bVisuBusy=FALSE) THEN
			bStartVisu:=FALSE;
			IF bVisuErr=FALSE THEN
				iState:=0;
			ELSE
				iState:=-3;
			END_IF
		END_IF
	1:	// Sűrített levegő bekapcsolása; hegesztő, TCP init
		MAIN.bLevego:=bLevego;
		GVL.bBiztonsagiZarBe:=TRUE;
		iStateHegeszto:=1;
		iStateTCP:=1;
		iState:=2;
	2:	// Hegesztőfejek + végmérő alapállása
		IF (MAIN.bLevegoOK=TRUE) THEN
			iStateHegesztoFejek:=1;
			iStateVegmero:=1;
			iStateHimba:=1;
			VEGMERO.bLezertakaro:=FALSE;
			iState:=3;
		END_IF
	3:	// Tengelyek indítása
		IF (bRobotKesz=TRUE) AND (bHegesztoFejekKesz=TRUE) AND (bVegmeroKesz=TRUE) AND (bHimbaKesz=TRUE) AND (bKameraKesz=TRUE) THEN
			iStateNTCTengely:=1;
			iStatePt1000Tengely:=1;
			iState:=4;
		END_IF
	4:	// Folyamatok ellenőrzése; befejezés
		IF (bHegesztoKesz=TRUE) AND (bNTCTengelyKesz=TRUE)
			AND (bPt1000TengelyKesz=TRUE) AND (VEGMERO.bLezertakaroZarva=TRUE)
			AND (GVL.bProductTypeOK=TRUE) THEN
			iState:=5;
			GVL.bSystemStarted:=TRUE;
			GVL.bSystemNotStarted:=FALSE;
		END_IF
	// RESET-elés
	10:
		MAIN.bLevego:=FALSE;
		GVL.bJozsiServo:=FALSE;
		GVL.bPistiServo:=FALSE;
		HEGESZTOK.bHegesztoMitStromOut:=FALSE;
		KAMERAREMOTE.bKameraSetOffline:=FALSE;
		KAMERAREMOTE.bKameraTriggerEN:=FALSE;
		KAMERAREMOTE.bKameraTrigger:=FALSE;
		iStateHegeszto := 0;		// Max 3
		iStateTCP := 0;				// Max 5
		iStateLezer := 0;			// Max 4
		iStateRobot := 0;			// Max 8
		iStateKamera := 0;			// Max 5
		iStateHegesztoFejek := 0;	// Max 3
		iStateVegmero := 0;			// Max 3
		iStateNTCTengely := 0;		// Max 5
		iStatePt1000Tengely := 0;	// Max 5
		iStateHimba := 0;			// Max 3
		bHegesztoKesz := FALSE;
		bTCPKesz := FALSE;
		bLezerKesz := FALSE;
		bRobotKesz := FALSE;
		bKameraKesz := TRUE;
		bHegesztoFejekKesz := FALSE;
		bVegmeroKesz := FALSE;
		bHimbaKesz := FALSE;
		bNTCTengelyKesz := FALSE;
		bPt1000TengelyKesz := FALSE;
		iKeszenletFoka := 0;
		iState:=11;
	11:
		GVL.bSystemStarted:=FALSE;
		GVL.bSystemNotStarted:=TRUE;
		iState:=0;
END_CASE

CASE iStateHegeszto OF
	1:	// Várakozás a hegesztő beindulására
		IF (HEGESZTOK.bHegesztoBereit=TRUE) THEN
			HEGESZTOK.bHegesztoMitStromOut:=TRUE;
			iStateHegeszto:=2;
		END_IF
	2:	// Hegesztőáram bekapcsolása
		IF (HEGESZTOK.bHegesztoBereit=TRUE) AND (HEGESZTOK.bHegesztoMitStromIn=TRUE) THEN
			iStateHegeszto:=3;	// Kész állapot
			bHegesztoKesz:=TRUE;
		END_IF
END_CASE

// TCP kapcsolatok reset-elése
CASE iStateTCP OF
	1:	// 1 ciklusig alsó szint a trigger jelnek
		bExecuteCloseAll:=FALSE;
		iStateTCP:=2;
	2:	// Felfutó él generálása a CloseAllSocket indításához
		bExecuteCloseAll:=TRUE;
		iStateTCP:=3;
	3:	// Várakozás, hogy elinduljon a CloseAllSocket()
		IF bCloseAllBusy=TRUE THEN
			iStateTCP:=4;
		END_IF
	4:	// Várakozás, amíg a CloseAllSocket() dolgozik
		IF bCloseAllBusy=FALSE THEN
			iStateLezer:=1;	// Lézer indítása
			iStateRobot:=1;	// Robot indítása
			iStateKamera:=1; //Pt Kamera indítása
//			TERMEKVALTAS.iState:=1; // Lézerprogram beállítása
			iStateTCP:=5;	// Kész állapot
			bTCPKesz:=TRUE;
		END_IF
END_CASE

// Pt Kamera indítása
CASE iStateKamera OF
	1: // Kamera online állapotba állítás, ha estleg még nem lenne
		KAMERAREMOTE.bKameraSetOffline:=FALSE;
		KAMERAREMOTE.bKameraTriggerEN:=FALSE;
		KAMERAREMOTE.bKameraTrigger:=FALSE;
		KameraProcess.bKameraRun:=TRUE;
		iStateKamera:=2;
	2: // Ha megjön az online jel, továbblépünk, különben várunk
		IF KAMERAREMOTE.bKameraOnline=TRUE THEN
			iStateKamera:=3;
		END_IF
	3: // Trigger EN jel küldése
		KAMERAREMOTE.bKameraTriggerEN:=TRUE;
		iStateKamera:=4;
	4: // Ha megjön a Trigger Ready jel, kész vagyunk
		IF KAMERAREMOTE.bKameraTriggerReady=TRUE THEN
			KameraProcess.bKameraRun:=FALSE;
			bKameraKesz:=TRUE;
			iStateKamera:=5; // Kész állapot
		END_IF
END_CASE

// Robot alaphelyzetbe
CASE iStateRobot OF
	1:	// Ajtók ellenőrzése
		IF GVL.bBiztonsagiFold=FALSE AND GVL.bBiztonsagiTap=TRUE THEN
			bStartDelay:=TRUE;
			iStateRobot:=2;
		END_IF
	2:	// Robotkommunikáció megnyitása
		IF bDelayEnd=TRUE THEN
			RobotProcess.s_InRobotCommand:='INIT';
			iStateRobot:=3;
		END_IF
	3:	//	Várakozás a robot válaszára
		IF ROBOTCOMMAND.sRobotResult='STATUSZ' THEN
			iStateRobot:=4;
		END_IF
	4:	// Robotpozíció ellenőrzése
		IF GVL.stRobotStatusz.rZ>-110 THEN
			iStateRobot:=7;
		ELSE
			RobotProcess.s_InRobotTCPCommand := 'HOME';
			iStateRobot:=5;
		END_IF
	5:	// Várakozás a robot HOME műveletének elkezdésére
		IF ROBOTCOMMAND.sRobotResult='' THEN
			iStateRobot:=6;
		END_IF
	6: // Várakozás a robot HOME műveletének végére
		IF ROBOTCOMMAND.sRobotResult='HOME' THEN
			iStateRobot:=7;
		END_IF
	7: // Várakozás a robot HOME műveletének végére
		iStateRobot:=8;	// Kész állapot
		bRobotKesz:=TRUE;
END_CASE

// Lézer státusz lekérdezése
CASE iStateLezer OF
	1:	// Státusz lekérdezése
		Laser.s_InCommand:='GETSTATUS';
		iStateLezer:=2;
	2:	//	Várakozás a lézer kézsenlétére
		IF Laser.s_Result='READY' THEN
			iStateLezer:=3;
		ELSIF Laser.s_Result='NOT_READY' THEN
			iStateLezer:=1;
		END_IF
	3:	// Jelenlegi beállított teljesítmény lekérdezése
		Laser.s_InCommand:='GETINTENSITY';
		bLezerKesz:=TRUE;
		iStateLezer:=4;		//Kész állapot
END_CASE

CASE iStateHegesztoFejek OF
	1:	// Minden hegesztőfej visszahúzása, szervók bekapcsolása
		HEGESZTOK.nHegesztoNum:=0;
		iStateHegesztoFejek:=2;
	2:	// Várakozás, hogy szabaddá váljon a kocsik útja
		IF	(GVL.bHegeszto1BalFent AND GVL.bHegeszto1JobbFent // 1. hegesztőfej visszahúzva
			AND GVL.bHegeszto2FentBent AND GVL.bHegeszto2LentBent // 2. hegesztőfej visszahúzva
			AND GVL.bHegeszto3Fent) THEN // 3. hegesztőfej visszahúzva
			iStateHegesztoFejek:=3;	// Kész állapot
			bHegesztoFejekKesz:=TRUE;
		END_IF
END_CASE

CASE iStateHimba OF
	1: //Himba vissza
		HIMBA.s_InCommand:='RESET';
		iStateHimba:=2;
	2: //Várakozás a Himba visszhúzódására
		IF HIMBA.s_InCommand='' THEN
			iStateHimba:=3;		//Kész állapot
			bHimbaKesz:=TRUE;
		END_IF
END_CASE

CASE iStateVegmero OF
	1:	// Minden hegesztőfej visszahúzása, szervók bekapcsolása
		VEGMERO.s_InCommand:='RESET';
		iStateVegmero:=2;
	2:	// Várakozás, hogy szabaddá váljon a kocsik útja
		IF	(VEGMERO.s_InCommand='') THEN 
			iStateVegmero:=3;	// Kész állapot
			bVegmeroKesz:=TRUE;
		END_IF
END_CASE

CASE iStateNTCTengely OF
	1:	// Várakozás, hogy szabaddá váljon a kocsik útja
		IF	(bNTCTengely AND GVL.bPres1FelsoFent AND GVL.bPres1AlsoLent // 1. prés visszahúzva
			AND GVL.bPres2FelsoFent AND GVL.bPres2AlsoLent // 2. prés visszahúzva
			AND GVL.bHegeszto1BalFent AND GVL.bHegeszto1JobbFent // 1. hegesztőfej visszahúzva
			AND GVL.bHegeszto2FentBent AND GVL.bHegeszto2LentBent // 2. hegesztőfej visszahúzva
			AND GVL.stRobotStatusz.rZ>-111.0) THEN// mérőtűk visszahúzva és robot fent
			iStateNTCTengely:=2;
		END_IF
(*	2: // NTC tengely 
		IF (JOZSITENGELY.bAxisReady = TRUE) THEN
			GVL.bJozsiServo:=bNTCTengely;
			iStateNTCTengely:=3;
		END_IF
	3:	IF JOZSITENGELY.bAxisOn THEN
			JOZSITENGELY.sJozsiAxisCommand:='HOME'; // 1. fázis kocsijának home-ba küldése
			iStateNTCTengely:=4;
		END_IF*)
	2:	// Home-ba küldés
		JOZSITENGELY.sJozsiAxisCommand:='HOME';
		iStateNTCTengely:=3;
	3: // NTC tengely 
		IF (JOZSITENGELY.bAxisReady = TRUE) THEN
			GVL.bJozsiServo:=TRUE;
			iStateNTCTengely:=4;
		END_IF
	4:	// Várakozás a tengely home-ba érkezésére
		IF (JOZSITENGELY.sJozsiAxisCommand='') AND (JOZSITENGELY.bHomeReady=TRUE) THEN
			iStateNTCTengely:=5;		//Kész állapot
			bNTCTengelyKesz:=TRUE;
		END_IF
END_CASE

CASE iStatePt1000Tengely OF
	1:	// Várakozás, hogy szabaddá váljon a kocsik útja
		IF	(bPt1000Tengely AND GVL.bHegeszto3Fent AND GVL.bKappepresFent // 3. hegesztőfej és Kappeprés visszahúzva
			AND VEGMERO.bMerotukBent AND GVL.stRobotStatusz.rZ>-111.0) THEN // mérőtűk visszahúzva és robot fent
			iStatePt1000Tengely:=2;
		END_IF
(*	2: // NTC tengely 
		IF (PISTITENGELY.bAxisReady = TRUE) THEN
			GVL.bPistiServo:=bNTCTengely;
			iStatePt1000Tengely:=3;
		END_IF
	3:	IF PISTITENGELY.bAxisOn THEN
			PISTITENGELY.sPistiAxisCommand:='HOME'; // 1. fázis kocsijának home-ba küldése
			iStatePt1000Tengely:=4;
		END_IF*)
	2: 
		PISTITENGELY.sPistiAxisCommand:='HOME'; // Home-ba küldés
		iStatePt1000Tengely:=3;
	3: // NTC tengely 
		IF (PISTITENGELY.bAxisReady = TRUE) THEN
			GVL.bPistiServo:=bNTCTengely;
			iStatePt1000Tengely:=4;
		END_IF
	4:	// Várakozás a tengely home-ba érkezésére
		IF (PISTITENGELY.sPistiAxisCommand='') AND (PISTITENGELY.bHomeReady=TRUE) THEN
			iStatePt1000Tengely:=5;		//Kész állapot
			bPt1000TengelyKesz:=TRUE;
		END_IF
END_CASE

iKeszenletFoka:=REAL_TO_INT(100*INT_TO_REAL(iStateHegeszto
				+iStateTCP
				+iStateLezer
				+iStateRobot
				+iStateKamera
				+iStateHegesztoFejek
				+iStateVegmero
				+iStateHimba
				+iStateNTCTengely
				+iStatePt1000Tengely)/44);

CASE iState2 OF
		1:	// Időpont beolvasása
			bStartGetTime:=TRUE;
			bStartWait:=TRUE;
			iState2:=2;
		2:	// Várakozás a busy jelre
			IF bGetTimeBusy=TRUE THEN
				iState2:=3;
			END_IF
		3:	// Várakozás az időpont beolvasás befejeztére
			IF bGetTimeBusy=FALSE THEN
				bStartGetTime:=FALSE;
				iState2:=4;
			END_IF
		4:	// Időpont beolvasás sikerességének vizsgálata
			IF bGetTimeError=FALSE THEN
				iState2:=5;
			ELSE
				iState2:=1;
			END_IF
		5:	// Szövegek előállítása (pl. a rendszeridőből)
			GVL.sYear:=WORD_TO_STRING(tstDateTime.wYear);
			GVL.sMonth:=WORD_TO_STRING(tstDateTime.wMonth);
			IF tstDateTime.wMonth<10 THEN
				GVL.sMonth:=CONCAT('0',GVL.sMonth);
			END_IF	
			GVL.sDay:=WORD_TO_STRING(tstDateTime.wDay);
			IF tstDateTime.wDay<10 THEN
				GVL.sDay:=CONCAT('0',GVL.sDay);
			END_IF	
			GVL.sHour:=WORD_TO_STRING(tstDateTime.wHour);
			IF tstDateTime.wHour<10 THEN
				GVL.sHour:=CONCAT('0',GVL.sHour);
			END_IF	
			GVL.sMinute:=WORD_TO_STRING(tstDateTime.wMinute);
			IF tstDateTime.wMinute<10 THEN
				GVL.sMinute:=CONCAT('0',GVL.sMinute);
			END_IF	
			GVL.sSecond:=WORD_TO_STRING(tstDateTime.wSecond);
			IF tstDateTime.wSecond<10 THEN
				GVL.sSecond:=CONCAT('0',GVL.sSecond);
			END_IF	
			GVL.sDateTime:=CONCAT(GVL.sYear,
							CONCAT('.',
							CONCAT(GVL.sMonth,
							CONCAT('.',
							CONCAT(GVL.sDay,
							CONCAT('.',
							CONCAT('  ',
							CONCAT(GVL.sHour,
							CONCAT(':',
							CONCAT(GVL.sMinute,
							CONCAT(':',GVL.sSecond)))))))))));
			iState2:=6;
		6:	IF bIdoLejart=TRUE THEN
				bStartWait:=FALSE;
				iState2:=1;
			END_IF
END_CASE

// Visualization indítása
FB_Start_Visu(
					NETID:='',
					PATHSTR:='C:\TwinCAT\3.1\Components\Plc\Tc3PlcHmi\Tc3PlcHmi.exe',
					DIRNAME:='C:\637\',
					COMNDLINE:='',
					START:=bStartVisu,
					TMOUT:=T#30S,
					BUSY => bVisuBusy,
					ERR => bVisuErr,
					ERRID => nVisuErr
					);

CloseAllSocket(
			sSrvNetId:= '', 
			bExecute:= bExecuteCloseAll, 
			tTimeout:= T#2000MS, 
			bBusy=> bCloseAllBusy, 
			bError=> bCloseAllError, 
			nErrId=> nCloseAllError);

GetTime(
		NETID:='',
		START:=bStartGetTime,
		TMOUT:=T#1S,
		BUSY=>bGetTimeBusy,
		ERR=>bGetTimeError,
		ERRID=>nGetTimeError,
		TIMESTR=>tstDateTime
		);

TDelay(IN:=bStartDelay, PT:=T#1S, Q=> bDelayEnd);

WAIT(IN:=bStartWait,PT:=T#100MS,Q=>bIdoLejart,ET=>);

FB_ShutDown(
			NETID:='',
			DELAY:=0,
			START:=bStartShutDown,
			TMOUT:=T#1M,
			BUSY =>,
			ERR => ,
			ERRID =>
			);

FB_RestartSystem(NETID:='',
				 RESTART:=bRestart,
				 TMOUT:=T#10S,
				 BUSY => bRestartBusy,
				 ERR => bRestartErr,
				 ERRID => nRestartErr);

END_PROGRAM

// ---- POUs/PISTI/Components/VEGMERO.TcPOU
PROGRAM VEGMERO
VAR_INPUT
	s_InCommand : STRING := '';
	s_InCommandParam1 : STRING := '';
	s_InCommandParam2 : STRING := '';
	s_InCommandParam3 : STRING := '';
	s_InCommandParam4 : STRING := '';
	s_InCommandParam5 : STRING := '';
	bLezertakaro AT %Q*: BOOL;
	iState : INT := 0;
END_VAR
VAR_OUTPUT
	n_OutErrId: UINT;
END_VAR
VAR
	//Platni
	bPlatniFelLe AT %Q*: BOOL;
	bPlatniBalraJobbra AT %Q*: BOOL;
	bHutesOn AT %Q*: BOOL;
	bPlatniFent AT %I*: BOOL;
	bPlatniLent AT %I*: BOOL;
	bNagyFeszMerotuLent AT %I*: BOOL;
	bPlatniBalon AT %I*: BOOL;
	bPlatniJobbon AT %I*: BOOL;
	bLezertakaroNyitva AT %I*: BOOL;
	bLezertakaroZarva AT %I*: BOOL;
	bHutes: BOOL:=FALSE;
	bAutoHutes: BOOL;
	bKeziHutes: BOOL;
	bHutesTiltas: BOOL := TRUE;
	tHutes: TIME := T#1S;
	TP_hutes: TP;
	
	
	//Merotuk
	bMerotukBeKi AT %Q*: BOOL;
	bMerotukBent AT %I*: BOOL;
	bMerotukKint AT %I*: BOOL;
	bRL_ISOL AT %Q*: BOOL;
	b600VBe AT %Q*: BOOL;
	PT_SOKK48V AT %Q*: BOOL;
	U12V AT %I*: INT;
	U600VExt AT %I*: INT;
	U600V AT %I*: INT;
	UISOL AT %I*: INT;
	PTRES AT %I*: INT;
	NTRES AT %I*: INT;
	NTRES2 AT %I*: INT;
	U48V AT %I*: INT;
	
	
	//FedelLecsukásÉrzékelő
	bFedelNyitva AT %I*: BOOL;
	
	//Hőszenzor
	iHorzekelo AT %I*: INT;
	
	//Értékek
	U12V_TRANS : REAL := 0;
	U600VExt_TRANS : REAL := 0;
	U600V_TRANS : REAL := 0;
	UISOL_TRANS : REAL := 0;
	PTRES_TRANS : REAL := 997.8/6617.5; // Rcal/Rcal_PTDIG: a teljes rendszer átvitele!
	NTRES_TRANS : REAL := 9955/16464; // Rcal/Rcal_NTC1DIG: a teljes rendszer átvitele!
	NTRES2_TRANS : REAL := 9955/16391; // Rcal/Rcal_NTC2DIG: a teljes rendszer átvitele!
	U48V_TRANS : REAL := 48.11/28640; // 48V_mert/48V_DIG
	PTRES_SCALE : REAL := 997.8/6617.5; // Rcal/Rcal_PTDIG: a teljes rendszer átvitele!
	NTRES_SCALE : REAL := 9955.0/16464; // Rcal/Rcal_NTC1DIG: a teljes rendszer átvitele!
	NTRES2_SCALE : REAL := 9955.0/16391; // Rcal/Rcal_NTC2DIG: a teljes rendszer átvitele!
	U48V_SCALE : REAL := 48.11/28640; // 48V_mert/48V_DIG
	U12V_SCALE : REAL := 12.114/19101; // 48V_mert/48V_DIG
	U48V_CAL : REAL;
	U12V_CAL : REAL;
	rHoerzekelo_TRANS : REAL := 0;
	PTRES_OC : REAL :=4800;
	NTRES_OC : REAL :=18000;
	
	//Kalkulációhoz
	PTRES_AMPLIFIER : REAL := 4.05;//2.0121/0.5012; //PT1000 erősítő értéke
	NTCRES_AMPLIFIER : REAL := 1.0001;//5.049/5.039; //NTC erősítő értéke
	NTCRES2_AMPLIFIER : REAL := 1.0132;//5.080/5.014; //NTC erősítő értéke
	PTRES_CURRENT : REAL := 0.5005/1005;//0.5mA-os áramgenerátor, feltételezhetően
	NTCRES_CURRENT : REAL := 5.041/10025;//0.5mA-os áramgenerátor, feltételezhetően
	NTCRES2_CURRENT : REAL := 5.014/9955;//0.5mA-os áramgenerátor, feltételezhetően
	PTRES_CALC : REAL := 0.0;
	PTRES_MIN : REAL := 0.0;
	PTRES_MAX : REAL := 0.0;
	NTCRES_MIN : REAL := 0.0;
	NTCRES_MAX : REAL := 0.0;
	NTCRES2_MIN : REAL := 0.0;
	NTCRES2_MAX : REAL := 0.0;
//	PTRES_SOKK_MAX : REAL := 2000.0;
	PTRES_MAXIdoallando : REAL := 0.0;
	NTRES_CALC : REAL := 0.0;
	NTRES2_CALC : REAL := 0.0;
	NTCTEMP_MAX : REAL := 0.0;
	NTCTEMP_MIN : REAL := 0.0;
	NTCTEMP_NOM : REAL := 0.0;
	NTCTEMP2_MAX : REAL := 0.0;
	NTCTEMP2_MIN : REAL := 0.0;
	NTCTEMP2_NOM : REAL := 0.0;
	ISOLRES_CALC : REAL := 0.0;
	fb_GetPT1000MinMaxResFromTemp : fb_GetPT1000MinMaxResFromTemp;
//	rTempMax : REAL := 300.0;	// Fűtőtömb hőmérséklete
//	tIdoallandoMax : TIME :=T#6S;
//	rIdoallandoMax : REAL :=6;
//	rISOL_MAX : REAL := 0.97;
	
	//Eredmények
	bFEDEL_ELLENORIZVE : BOOL := FALSE;
	bPTRES_OK : BOOL := FALSE;
	bPTRES_MERVE : BOOL;
	bNTCRES_OK : BOOL := FALSE;
	bNTCRES2_OK : BOOL := FALSE;
	bNTCRES_MERVE : BOOL;
	bNTCRES2_MERVE : BOOL;
	bISOL_OK : BOOL := FALSE;
	bISOL_MERVE : BOOL;
	bIDOALLANDO_OK : BOOL := FALSE;
	bIDOALLANDO_MERVE : BOOL;
	bSOKK_OK : BOOL := FALSE;
	bSOKK_MERVE : BOOL;
	rPTRES: REAL := 0.0;
	rNTCRES: REAL := 0.0;
	rNTCRES2: REAL := 0.0;
	rISOL: REAL := 0.0;
	aPTRES: ARRAY[0..9] OF REAL;
	aNTCRES: ARRAY[0..9] OF REAL;
	aNTCRES2: ARRAY[0..9] OF REAL;
	aTEMP: ARRAY[0..9] OF REAL;
	aISOL: ARRAY[0..39] OF REAL;
	tIdoallando : TIME := T#0MS;
	atIdoallando : ARRAY[0..600] OF TIME;
	raIdoallandoIdo : ARRAY[0..600] OF REAL;
	arIdoallandoPTTEMP : ARRAY[0..600] OF REAL;
	rPTTEMP : REAL;
	raIdoallandoPTR : ARRAY[0..500] OF REAL;
//	raTemperatureCurve : ARRAY[0..1,0..2000] OF REAL;
	
	//INTERNAL
	nI: INT := 0;
	s_InLCommand : STRING := '';
	T_Ticker : TON;
	bTickerEnable : BOOL := FALSE;
	tTickerTimeCsatlakozas : TIME := T#1000MS;
	tTickerTime600VKijutas : TIME := T#1000MS;
	tTickerTimeIdoallando : TIME := T#6000MS;
	tTickerTimeSokk : TIME := T#2000MS;
	tTickerTimeSokkEll : TIME := T#2000MS;
	tTickerTime : TIME := T#300MS;
	bTickerQ : BOOL := FALSE;
	tTickerET : TIME := T#0MS;
	bFolyamatos : BOOL := FALSE;
	bMasodikEllMeres : BOOL;
	
	rTemp: REAL;

	// Mérő kapcsolás megnyitása
	FB_Start_Schematic: NT_StartProcess;
	bStartSchematic: BOOL;
	bSchematicBusy: BOOL;
	bSchematicErr: BOOL;
	nSchematicErr: UDINT;
	iState2: INT;
	rIdoallandoPTTEMP: REAL;
	
END_VAR

U12V_TRANS := U12V/3276.7;
U600VExt_TRANS := U600VExt/3276.7;
U600V_TRANS := U600V/3276.7;
UISOL_TRANS := UISOL/3276.7;
// PTRES_TRANS := PTRES/3276.7;
// NTRES_TRANS := NTRES/3276.7;
// NTRES2_TRANS := NTRES2/3276.7;
// U48V_TRANS := U48V/3276.7;
U48V_CAL := U48V*U48V_SCALE;
U12V_CAL := U12V*U12V_SCALE;
rHoerzekelo_TRANS := (INT_TO_REAL(iHorzekelo)/100);
// PTRES_CALC := (PTRES_TRANS/PTRES_AMPLIFIER) / PTRES_CURRENT*0.995; // A 0.995 egy korrekciós tényező
PTRES_CALC := PTRES*PTRES_SCALE;
NTRES_CALC := NTRES*NTRES_SCALE;
NTRES2_CALC := NTRES2*NTRES2_SCALE;

(*IF s_InCommand <>'' AND s_InCommand[0] <> '_' AND iState = 0 THEN
	IF (s_InCommand <>'RESET') THEN
		s_InLCommand := s_InCommand;
		n_OutErrId := 0;
		iState := 1;
	ELSE
		s_InLCommand := '';
		s_InCommand := '';
	END_IF
	bMasodikEllMeres:=FALSE;
	bPTRES_OK := FALSE;
	bNTCRES_OK := FALSE;
	bSOKK_OK := FALSE;
	bISOL_OK := FALSE;
END_IF*)
CASE iState OF
	0:	// Parancsra várás
		IF s_InCommand <>'' AND LEFT(s_InCommand,1) <> '_' THEN
			IF (s_InCommand <>'RESET') THEN
				s_InLCommand := s_InCommand;
				n_OutErrId := 0;
				iState := 1;
			ELSE
				iState:=20100;
			END_IF
			bMasodikEllMeres:=FALSE;
			bFEDEL_ELLENORIZVE:=FALSE;
			bPTRES_MERVE := FALSE;
			GVL.bPTResOK := FALSE;
			bNTCRES_MERVE := FALSE;
			GVL.bNTCResOK := FALSE;
			bISOL_MERVE := FALSE;
			GVL.bIsolOK := FALSE;
			bIDOALLANDO_MERVE := FALSE;
			GVL.bTimeConstOK := FALSE;
			bSOKK_MERVE := FALSE;
			GVL.bShockOK := FALSE;			
		END_IF
	1:	// Alaphelyzet ellenőrzése
		IF (bMerotukBent = TRUE AND bMerotukKint = FALSE
			AND bPlatniLent = FALSE AND bNagyFeszMerotuLent = FALSE
			AND bPlatniFent = TRUE) THEN
			n_OutErrId := 0;
			iState := 2;
		ELSIF MAIN.bLevegoOK=FALSE THEN
			n_OutErrId:=5;
		ELSIF (bMerotukBent = FALSE) THEN
			n_OutErrId:=87;
		ELSIF bMerotukKint = TRUE THEN
			n_OutErrId:=86;
		ELSIF bPlatniLent = TRUE THEN
			n_OutErrId:=84;
		ELSIF bNagyFeszMerotuLent = TRUE THEN
			n_OutErrId:=112;
		ELSIF bPlatniFent = FALSE THEN
			n_OutErrId:=81;
		END_IF
	2:	// Mérőtűk kitolása
		bMerotukBeKi := TRUE;
		iState := 3;
	3:	// Várakozás a mérőtűk érkezésére
		IF (bMerotukBent = FALSE AND bMerotukKint = TRUE) THEN
			n_OutErrId := 0;
			iState := 4;
		ELSIF MAIN.bLevegoOK=FALSE THEN
			n_OutErrId:=5;
		ELSIF bMerotukBent = TRUE THEN
			n_OutErrId:=88;
		ELSIF bMerotukKint = FALSE THEN
			n_OutErrId:=85;
		END_IF
	4:	// További várakozás indítása a mérőtűk megérkezése után
		IF bTickerEnable = TRUE THEN
			bTickerEnable := FALSE;
		ELSE
			bTickerEnable := TRUE;
			IF (s_InCommand='ETALONMERES') THEN	
				tTickerTime := T#10000MS; //tTickerTimeCsatlakozas;
			ELSE
				tTickerTime := T#1000MS;
			END_IF
			iState := 5;
		END_IF
	5:	// Várakozási idő letelte
		IF bTickerQ = TRUE THEN
			bTickerEnable := FALSE;
//			iState := 800;
			iState := 6;
		END_IF
	6:	// Csatlakozó fedél ellenőrzése
		GVL.bFedelOK:=(*NOT *)bFedelNyitva;
			bFEDEL_ELLENORIZVE:=TRUE;
		IF ((GVL.bFedelOK=(*FALSE*)TRUE) OR (GVL.iSelectedProductType>8)) OR (s_InCommand='ETALONMERES') THEN
			iState := 800;
		ELSE
			s_InCommand:='_FEDELNYITVA';
			iState:=20000;
		END_IF
		
	//	Ellenállásmérés
	30:	// Inicializálás
		nI := 0;
		bHutes:=TRUE;
		IF bMasodikEllMeres=FALSE THEN	// Ha nem volt előtte sokkolás, ...
			iState := 33;
		ELSE
			iState := 31;
		END_IF			
	31: // Sokkolás utáni várakozás indítása
		IF bTickerEnable = TRUE THEN
			bTickerEnable := FALSE;
		ELSE
			bTickerEnable := TRUE;
			tTickerTime := tTickerTimeSokkEll;
			iState := 32;
		END_IF
	32: // Letelt a sokkolás utáni várakozási idő
		IF bTickerQ = TRUE THEN
			iState := 33;
			bTickerEnable := FALSE;
		END_IF
	33: // Várakozás a hűtés végére
		IF (bHutesOn=FALSE) THEN
			bHutes:=FALSE;
			iState:=34;
		END_IF
	34:	// nI. mért érték beolvasása
		aPTRES[nI] := PTRES_CALC;
		aNTCRES[nI] := NTRES_CALC;
		aNTCRES2[nI] := NTRES2_CALC;
		aTEMP[nI] := rHoerzekelo_TRANS;
		nI := nI + 1;
		iState := 35;
	35:	// Ha mért már 10 értéket, akkor a 10 érték átlagolása
		IF nI > 9 THEN
			rPTRES := 0;
			rNTCRES := 0;
			rNTCRES2 := 0;
			rTemp := 0;
			FOR nI := 0 TO 9 BY 1 DO
				rPTRES := rPTRES + aPTRES[nI];
				rNTCRES := rNTCRES + aNTCRES[nI];
				rNTCRES2 := rNTCRES2 + aNTCRES2[nI];
				rTemp := rTemp + aTEMP[nI];
			END_FOR
			rNTCRES := rNTCRES / 10;
			rNTCRES2 := rNTCRES2 / 10;
			rPTRES := rPTRES / 10;
			rTemp := rTemp / 10;
			iState := 36;
		ELSE
			iState := 34;
		END_IF
	36:	// Ellenállásmérési eredmények kiértékelése
//		fb_GetPT1000MinMaxResFromTemp(rTemp:= rHoerzekelo_TRANS, rResMin=> PTRES_MIN, rResMax=> PTRES_MAX);
		PTRES_MIN:=f_GetPtMinR(rTemp:=rTemp);
		PTRES_MAX:=f_GetPtMaxR(rTemp:=rTemp);
		IF GVL.iCurrentProductType>=0 THEN
			NTCRES_MIN:=f_GetNTCMinR(rTemp:=rTemp,nProd:=0,rNTCDev:=GVL.rNTCDev);
			NTCRES_MAX:=f_GetNTCMaxR(rTemp:=rTemp,nProd:=0,rNTCDev:=GVL.rNTCDev);
		ELSE
			NTCRES_MIN:=f_GetNTCMinR(rTemp:=rTemp,nProd:=0,rNTCDev:=7);
			NTCRES_MAX:=f_GetNTCMaxR(rTemp:=rTemp,nProd:=0,rNTCDev:=7);
		END_IF
		NTCTEMP_MIN := f_GetNTCMinTempFromRes(rNTCRES);
		NTCTEMP_MAX := f_GetNTCMaxTempFromRes(rNTCRES);
		NTCTEMP_NOM := f_GetNTCNomTempFromRes(rNTCRES);
		IF GVL.iCurrentProductType>=0 THEN
			NTCRES2_MIN:=f_GetNTCMinR(rTemp:=rTemp,nProd:=0,rNTCDev:=GVL.rNTC2Dev);
			NTCRES2_MAX:=f_GetNTCMaxR(rTemp:=rTemp,nProd:=0,rNTCDev:=GVL.rNTC2Dev);
		ELSE
			NTCRES2_MIN:=f_GetNTCMinR(rTemp:=rTemp,nProd:=0,rNTCDev:=7);
			NTCRES2_MAX:=f_GetNTCMaxR(rTemp:=rTemp,nProd:=0,rNTCDev:=7);
		END_IF
		NTCTEMP2_MIN := f_GetNTCMinTempFromRes(rNTCRES2);
		NTCTEMP2_MAX := f_GetNTCMaxTempFromRes(rNTCRES2);
		NTCTEMP2_NOM := f_GetNTCNomTempFromRes(rNTCRES2);
		IF (bMasodikEllMeres=FALSE) THEN
			rPTTEMP:=f_GetPTTEMPFromRES(PTRES_CALC); // Időállandó görbe állandó szobahőm.-re
			FOR nI:=0 TO 600 DO
				arIdoallandoPTTEMP[nI] := rPTTEMP;
			END_FOR
			GVL.rTemp:=rHoerzekelo_TRANS;
			GVL.rPtRes:=rPTRES;
			bPTRES_MERVE := TRUE;
			IF PTRES_MIN<=rPTRES AND PTRES_MAX>=rPTRES THEN
				bPTRES_OK := TRUE;
			ELSE
				bPTRES_OK := FALSE;
			END_IF
			GVL.bPTResOK:=bPTRES_OK;
			IF bPTRES_OK=TRUE THEN
				GVL.iPTResQ:=1;
			ELSE			
				GVL.iPTResQ:=2;
			END_IF
			GVL.rNTCRes:=rNTCRES;
			IF NTCRES_MIN<=rNTCRES AND NTCRES_MAX>=rNTCRES THEN
				bNTCRES_OK := TRUE;
			ELSE
				bNTCRES_OK := FALSE;
			END_IF;
			bNTCRES_MERVE := TRUE;
			IF GVL.iSelectedProductType>8 THEN // 745 esetén
				GVL.rNTCRes2:=rNTCRES2;
				IF NTCRES2_MIN<=rNTCRES2 AND NTCRES2_MAX>=rNTCRES2 THEN
					bNTCRES2_OK := TRUE;
				ELSE
					bNTCRES2_OK := FALSE;
				END_IF
				bNTCRES2_MERVE := TRUE;
			ELSE
				rNTCRES2:=0;
				GVL.rNTCRes2:=0;
				bNTCRES2_MERVE := FALSE;
			END_IF;				
(*			IF NTCTEMP_MAX <= rHoerzekelo_TRANS AND NTCTEMP_MIN >= rHoerzekelo_TRANS THEN
				bNTCRES_OK := TRUE;
			ELSE
				bNTCRES_OK := FALSE;
			END_IF*)
			GVL.bNTCResOK:=bNTCRES_OK;
			IF bNTCRES_OK=TRUE THEN
				GVL.iNTCResQ:=1;
			ELSE	
				GVL.iNTCResQ:=2;
			END_IF
			GVL.bNTCRes2OK:=bNTCRES2_OK;
			IF bNTCRES2_OK=TRUE THEN
				GVL.iNTC2ResQ:=1;
			ELSE	
				GVL.iNTC2ResQ:=2;
			END_IF
			IF (rPTRES>PTRES_OC) OR (rNTCRES>NTRES_OC) THEN
				s_InCommand:='_SZAKADAS';
				s_InLCommand:='';
				iState:=20000;
			END_IF
		ELSE	// Ha volt előtte sokkolás
			bSOKK_MERVE := TRUE;
			IF GVL.PTRES_SOKK_MAX>=rPTRES THEN
				bSOKK_OK := TRUE;
			ELSE
				bSOKK_OK := FALSE;
			END_IF
			GVL.rPtResShock:=rPTRES;
			GVL.bShockOK:=bSOKK_OK;
			IF bSOKK_OK=TRUE THEN
				GVL.iShockQ:=1;
			ELSE
				GVL.iShockQ:=2;
			END_IF
		END_IF
		IF (s_InCommand='TELJESMERES') OR (s_InCommand='ETALONMERES') THEN
			iState := 800;
		ELSE				
			iState := 20000;
		END_IF
		
	//ÁTÜTÉS
	50:	// Platni fordítása szigetelésvizsgálathoz
		bPlatniBalraJobbra := TRUE;
		bRL_ISOL := TRUE;
		iState := 51;
	51:	// Várakozás a platni befordulására
		IF bPlatniBalon = TRUE AND bPlatniJobbon = FALSE THEN
			n_OutErrId := 0;
			iState := 54;
		ELSIF MAIN.bLevegoOK=FALSE THEN
			n_OutErrId:=5;
		ELSIF bPlatniBalon = FALSE THEN
			n_OutErrId:=107;
		ELSIF bPlatniJobbon = TRUE THEN
			n_OutErrId:=106;
		END_IF
	54:	// Szigetelés mérőtűk leeresztése
		bPlatniFelLe := TRUE;
		iState := 55;
	55:	// Várakozás a mérőtűk megérkezésére
		IF bPlatniFent = FALSE AND bNagyFeszMerotuLent = TRUE THEN
			n_OutErrId := 0;
			iState := 58;
		ELSIF MAIN.bLevegoOK=FALSE THEN
			n_OutErrId:=5;
		ELSIF bPlatniFent = TRUE THEN
			n_OutErrId:=82;
		ELSIF bNagyFeszMerotuLent = FALSE THEN
			n_OutErrId:=111;
		END_IF
	58:	// 600V rákapcsolása
		b600VBe := TRUE;
		iState := 59;
	59:	// 600V timeout indítása
		IF bTickerEnable = TRUE THEN
			bTickerEnable := FALSE;
		ELSE
			bTickerEnable := TRUE;
			tTickerTime := tTickerTime600VKijutas;
			iState := 60;
		END_IF
	60:	// Megjelent-e a 600V?	
		IF bTickerQ = TRUE OR U600V_TRANS>6 THEN
			bTickerEnable := FALSE;
			IF U600V_TRANS>6 THEN
				iState := 61;
			ELSE
				//Nem kapcsol be a 600V
				n_OutErrId := 197;
			END_IF
		END_IF
	61:	// Timeout időzítő törlése, újraindítása
		IF bTickerEnable = TRUE THEN
			bTickerEnable := FALSE;
		ELSE
			bTickerEnable := TRUE;
			tTickerTime := tTickerTime600VKijutas;
			iState := 62;
		END_IF
	62:	// Megjelent-e a 600V a Kappe-n? Ha a termék zárlatos, akkor sem jelenik meg a 600V.
		IF bTickerQ = TRUE OR U600VExt_TRANS > 4.5 OR UISOL_TRANS>GVL.rISOL_MAX THEN
			IF bTickerQ = FALSE THEN
				iState := 63;
			ELSE
				//Nem megy ki a 600V A kappéra
				n_OutErrId := 199;
			END_IF
			bTickerEnable := FALSE;
		END_IF
	63: // Szigetelés vizsgálat inicializálása
		nI := 0;
		iState := 64;
	64:	// Szigetelési érték olvasása
		aISOL[nI] := UISOL_TRANS;
		nI := nI + 1;
		iState := 65;
	65:	// Ha van már 40 mérés, akkor átlagolás
		IF nI > 39 THEN
			rISOL := 0;
			FOR nI := 0 TO 39 BY 1 DO
				rISOL := rISOL + aISOL[nI];
			END_FOR
			rISOL := rISOL / 40;
			iState := 66;
		ELSE
			iState := 64;
		END_IF
	66:	// Szigetelés vizsgálat kiértékelése
		bISOL_MERVE := TRUE;
		IF rISOL < GVL.rISOL_MAX THEN
			bISOL_OK := TRUE;
		ELSE //Átütéses			
			bISOL_OK := FALSE;
		END_IF
		iState := 20100;
		GVL.bIsolOK:=bISOL_OK;
		IF bISOL_OK=TRUE THEN
			GVL.iIsolQ:=1;
		ELSE	
			GVL.iIsolQ:=2;
		END_IF

	// Időállandó mérése		
	100: // Ha a jelenlegi ellenállásérték nem haladja meg a várt végértéket, ...
//		fb_GetPT1000MinMaxResFromTemp(rTemp:= rHoerzekelo_TRANS, rResMin=> , rResMax=> PTRES_MAXIdoallando);
		rPTTEMP:=f_GetPTTEMPFromRES(PTRES_CALC); // Időállandó görbe állandó szobahőm.-re
		FOR nI:=0 TO 600 DO
			arIdoallandoPTTEMP[nI] := rPTTEMP;
		END_FOR
		PTRES_MAXIdoallando:=f_GetPtMaxR(rHoerzekelo_TRANS);
		IF PTRES_MAXIdoallando>=rPTRES THEN
			bPlatniBalraJobbra := FALSE;
			iState := 101;
		ELSE //Túl meleg PT1000
			iState := 20000;
		END_IF
	101: // Platni leengedése
		IF bPlatniBalon = FALSE AND bPlatniJobbon = TRUE THEN
			bPlatniFelLe := TRUE;
			n_OutErrId := 0;
			iState := 102;
		ELSIF MAIN.bLevegoOK=FALSE THEN
			n_OutErrId:=5;
		ELSIF bPlatniBalon = TRUE THEN
			n_OutErrId:=108;
		ELSIF bPlatniJobbon = FALSE THEN
			n_OutErrId:=105;
		END_IF
	102: // Várakozás a platni érkezésére
		IF bPlatniFent = FALSE AND bPlatniLent = TRUE THEN
			n_OutErrId := 0;
			iState := 103;
		ELSIF MAIN.bLevegoOK=FALSE THEN
			n_OutErrId:=5;
		ELSIF bPlatniFent = TRUE THEN
			n_OutErrId:=82;
		ELSIF bPlatniLent = FALSE THEN
			n_OutErrId:=83;
		END_IF
	103: // Időállandó mérés inicializálása
		nI:=0;
		iState := 104;
	104: // Timeout timer indítása (6s)
		IF bTickerEnable = TRUE THEN
			bTickerEnable := FALSE;
		ELSE
			bTickerEnable := TRUE;
			tTickerTime := tTickerTimeIdoallando;
			iState := 105;
		END_IF
	105: // Van-e timeout vagy túlfutás?
		IF bTickerQ = TRUE OR nI = 600 THEN
			bTickerEnable := FALSE;
			tIdoallando := T#6100MS;
			GVL.rTimeConst:=TIME_TO_REAL(tIdoallando)/1000;
			bIDOALLANDO_MERVE := TRUE;
			bIDOALLANDO_OK := FALSE;
			GVL.bTimeConstOK:=bIDOALLANDO_OK;
			iState := 108;
		ELSE	// Mérési pont felvétele, mentése
			atIdoallando[nI] := tTickerET;
			raIdoallandoIdo[nI] := TIME_TO_REAL(tTickerET)/1000.0;
//			raTemperatureCurve[0,nI] := TIME_TO_REAL(tTickerET)/1000.0;
			raIdoallandoPTR[nI]:=PTRES_CALC;
			rIdoallandoPTTEMP:=f_GetPTTEMPFromRES(PTRES_CALC);
			arIdoallandoPTTEMP[nI] := f_GetPTTEMPFromRES(PTRES_CALC);
//			raTemperatureCurve[1,nI] := f_GetPTTEMPFromRES(PTRES_CALC);
			iState := 106;
		END_IF
	106: // Leállási feltétel vizsgálata
		IF arIdoallandoPTTEMP[nI]>=((GVL.rTempMax-arIdoallandoPTTEMP[0])*0.63+arIdoallandoPTTEMP[0]) THEN
			iState := 107; // Leállás
			bTickerEnable := FALSE;
		ELSE
			nI:=nI+1;
			iState := 105; // Újabb mérési pont
		END_IF
	107: // Időállandó mérés kiértékelése
		tIdoallando := atIdoallando[nI]-atIdoallando[0];
		bIDOALLANDO_MERVE := TRUE;
		IF tIdoallando<REAL_TO_TIME(GVL.rIdoallandoMax*1000) THEN
			bIDOALLANDO_OK := TRUE;
		ELSE
			bIDOALLANDO_OK := FALSE;
		END_IF
		GVL.rTimeConst:=TIME_TO_REAL(tIdoallando)/1000;
		GVL.bTimeConstOK:=bIDOALLANDO_OK;
		IF bIDOALLANDO_OK=TRUE THEN
			GVL.iTimeConstQ:=1;
		ELSE	
			GVL.iTimeConstQ:=2;
		END_IF
		iState := 108;
	108: // Platni felemelése
		bPlatniFelLe := FALSE;
		iState:=109;
	109: // Várakozás a platni érkezésére
		IF bPlatniFent = TRUE AND bPlatniLent = FALSE THEN
			bPlatniBalraJobbra := TRUE;
			n_OutErrId := 0;
			iState := 110;
		ELSIF MAIN.bLevegoOK=FALSE THEN
			n_OutErrId:=5;
		ELSIF bPlatniFent = FALSE THEN
			n_OutErrId:=81;
		ELSIF bPlatniLent = TRUE THEN
			n_OutErrId:=84;
		END_IF
	110: // Várakozás a platni elfordulására
		IF bPlatniBalon = TRUE AND bPlatniJobbon = FALSE THEN
			n_OutErrId := 0;
			iState := 20200;
		ELSIF MAIN.bLevegoOK=FALSE THEN
			n_OutErrId:=5;
		ELSIF bPlatniBalon = FALSE THEN
			n_OutErrId:=107;
		ELSIF bPlatniJobbon = TRUE THEN
			n_OutErrId:=106;
		END_IF

	// Sokkolás	
	200: // 48V meglétének ellenőrzése
		IF U48V_CAL>47.5 THEN
			iState := 201;
		ELSE
			n_OutErrId := 201;
		END_IF
	201: // 48V rákapcsolása
		PT_SOKK48V := TRUE;
		iState := 202;
	202: // Sokkolás idejének indítása
		IF bTickerEnable = TRUE THEN
			bTickerEnable := FALSE;
		ELSE
			bTickerEnable := TRUE;
			tTickerTime := tTickerTimeSokk;
			iState := 203;
		END_IF
	203: // Letelt a sokkolás ideje
		IF bTickerQ = TRUE THEN
			iState := 204;
			bTickerEnable := FALSE;
		END_IF
	204: // 48V lekapcsolása
		PT_SOKK48V := FALSE;
		IF (s_InCommand='TELJESMERES') THEN
			iState := 800;
		ELSE				
			iState := 20000;
		END_IF

	// Ellenállás etalon mérése		
	300: // Etalonmérés inicializálása
		nI := 0;
		iState := 301;
	301: // Mérési pont felvétele
		aPTRES[nI] := PTRES_CALC;
		aNTCRES[nI] := NTRES_CALC;
		nI := nI + 1;
		iState := 302;
	302: // Megvan-e a 10 mérési pont?
		IF nI > 9 THEN
			rPTRES := 0;
			rNTCRES := 0;
			FOR nI := 0 TO 9 BY 1 DO
				rPTRES := rPTRES + aPTRES[nI];
				rNTCRES := rNTCRES + aNTCRES[nI];
			END_FOR
			rNTCRES := rNTCRES / 10;
			rPTRES := rPTRES / 10;
			iState := 303;
		ELSE
			iState := 301;
		END_IF
	303: // Etalonmérés kiértékelése
		fb_GetPT1000MinMaxResFromTemp(rTemp:= 0, rResMin=> PTRES_MIN, rResMax=> PTRES_MAX);
		NTCTEMP_MIN := f_GetNTCMinTempFromRes(rNTCRES);
		NTCTEMP_MAX := f_GetNTCMaxTempFromRes(rNTCRES);
		NTCTEMP_NOM := f_GetNTCNomTempFromRes(rNTCRES);
		IF PTRES_MIN<=rPTRES AND PTRES_MAX>=rPTRES THEN
			bPTRES_OK := TRUE;
		ELSE
			bPTRES_OK := FALSE;
		END_IF
		IF NTCTEMP_MAX <= 25 AND NTCTEMP_MIN >= 25 THEN
			bNTCRES_OK := TRUE;
		ELSE
			bNTCRES_OK := FALSE;
		END_IF
		iState := 20000;
		
	800: // Parancsértelmezés
		IF s_InCommand = 'TELJESMERES' THEN
			IF s_InLCommand = 'TELJESMERES' THEN
				s_InLCommand:='ELLENALLAS';
				bMasodikEllMeres:=FALSE;
			ELSIF s_InLCommand = 'ELLENALLAS' THEN
				s_InLCommand:='ATUTES';
			ELSIF s_InLCommand = 'ATUTES' THEN
				s_InLCommand:='IDOALLANDO';
			ELSIF s_InLCommand = 'IDOALLANDO' THEN
				s_InLCommand:='SOKK';
			ELSIF s_InLCommand = 'SOKK' THEN
				s_InCommand:='ELLENALLAS';
				s_InLCommand:='ELLENALLAS';
				bMasodikEllMeres:=TRUE;
			END_IF
		ELSIF s_InCommand = 'ETALONMERES' THEN
			IF s_InLCommand = 'ETALONMERES' THEN
				s_InLCommand:='ELLENALLAS';
				bMasodikEllMeres:=FALSE;
			ELSIF s_InLCommand = 'ELLENALLAS' THEN
				s_InLCommand:='ATUTES';
			ELSIF s_InLCommand = 'ATUTES' THEN
				s_InLCommand:='IDOALLANDO';
				s_InCommand:='IDOALLANDO';
			END_IF
		END_IF
		IF s_InLCommand = 'ELLENALLAS' THEN
//			bPTRES_OK := FALSE;
//			bNTCRES_OK := FALSE;
//			bSOKK_OK := FALSE;
			PTRES_CALC := 0;
			NTRES_CALC := 0;
			iState := 30;
		ELSIF s_InLCommand = 'ATUTES' THEN
//			bISOL_OK := FALSE;
			ISOLRES_CALC := 0;
			iState := 50;
		ELSIF s_InLCommand = 'IDOALLANDO' THEN
			tIdoallando := T#0MS;
			bIDOALLANDO_OK := FALSE;
			iState := 100;
		ELSIF s_InLCommand = 'SOKK' THEN
			iState := 200;
		ELSIF s_InLCommand = 'ELLENALLASETALON' THEN
//			bPTRES_OK := FALSE;
//			bNTCRES_OK := FALSE;
			PTRES_CALC := 0;
			NTRES_CALC := 0;
			iState := 300;
		ELSE
			iState := 20000;
		END_IF
		
	900:
		IF s_InLCommand = 'ELLENALLAS' THEN
			bPTRES_OK := FALSE;
			bNTCRES_OK := FALSE;
			PTRES_CALC := 0;
			NTRES_CALC := 0;
			iState := 30;
		ELSE
			iState := 901;
		END_IF
	901:
		IF s_InLCommand = 'ATUTES' THEN
			bISOL_OK := FALSE;
			ISOLRES_CALC := 0;
			iState := 50;
		ELSE
			iState := 902;
		END_IF
	902:
		IF s_InLCommand = 'IDOALLANDO' THEN
			tIdoallando := T#0MS;
			bIDOALLANDO_OK := FALSE;
			iState := 100;
		ELSE
			iState := 903;
		END_IF
	903:
		IF s_InLCommand = 'SOKK' THEN
			iState := 200;
		ELSE
			iState := 904;
		END_IF
	904:
		IF s_InLCommand = 'ELLENALLASETALON' THEN
			bPTRES_OK := FALSE;
			bNTCRES_OK := FALSE;
			PTRES_CALC := 0;
			NTRES_CALC := 0;
			iState := 300;
		ELSE
			iState := 20000;
		END_IF
		
	// Lecsatlakozás
	20000:
		bPlatniFelLe:=FALSE;
		bMerotukBeKi := FALSE;
		iState:=20005;
	20005:
		IF (bMerotukBent = TRUE AND bMerotukKint = FALSE) THEN
			IF LEFT(s_InCommand,1)<>'_' AND s_InCommand<>'RESET' THEN
				iState := 30000;
			ELSE
				iState := 0;
				s_InCommand:='';
			END_IF
			IF LEFT(s_InCommand,1)<>'_' THEN
				s_InCommand := '';
				s_InLCommand := '';
			END_IF
			n_OutErrId := 0;
		ELSIF MAIN.bLevegoOK=FALSE THEN
			n_OutErrId:=5;
		ELSIF bMerotukBent = FALSE THEN
			n_OutErrId:=87;
		ELSIF bMerotukKint = TRUE THEN
			n_OutErrId:=86;
		END_IF
		
	//Leállítási procedúrák
	//Izoláció leállítás
	20100:
		b600VBe := FALSE;
		iState := 20101;
	20101:
		IF U600V_TRANS<0.5 THEN
			n_OutErrId := 0;
			iState := 20102;
		ELSE
			n_OutErrId:=203;
		END_IF
	20102:
		bRL_ISOL := FALSE;
		bPlatniFelLe := FALSE;
		iState := 20103;
	20103:
		IF bPlatniLent = FALSE AND bNagyFeszMerotuLent = FALSE
			AND bPlatniFent = TRUE THEN
			n_OutErrId := 0;
			iState := 20104;
		ELSIF MAIN.bLevegoOK=FALSE THEN
			n_OutErrId:=5;
		ELSIF bPlatniLent = TRUE THEN
			n_OutErrId:=84;
		ELSIF bNagyFeszMerotuLent = TRUE THEN
			n_OutErrId:=112;
		ELSIF bPlatniFent = FALSE THEN
			n_OutErrId:=81;
		END_IF
	20104:
		bPlatniBalraJobbra := TRUE;
		iState := 20105;
	20105:
		IF bPlatniBalon = TRUE AND bPlatniJobbon = FALSE THEN
			IF (s_InCommand='TELJESMERES') OR (s_InCommand='ETALONMERES') THEN
				iState := 800;
			ELSE				
				iState := 20000;
			END_IF
			n_OutErrId := 0;
		ELSIF MAIN.bLevegoOK=FALSE THEN
			n_OutErrId:=5;
		ELSIF bPlatniBalon = FALSE THEN
			n_OutErrId:=107;
		ELSIF bPlatniJobbon = TRUE THEN
			n_OutErrId:=106;
		END_IF
		
	//Iőállandó leállítás
	20200:
		bPlatniFelLe := FALSE;
		iState := 20205;
	20205: // Várakozás a platni felemelkedésére
		IF (bPlatniLent = FALSE AND bNagyFeszMerotuLent = FALSE
			AND bPlatniFent = TRUE) THEN
			bPlatniBalraJobbra:=TRUE;
			n_OutErrId := 0;
			iState:=20210;
		ELSIF MAIN.bLevegoOK=FALSE THEN
			n_OutErrId:=5;
		ELSIF bPlatniLent = TRUE THEN
			n_OutErrId:=84;
		ELSIF bNagyFeszMerotuLent = TRUE THEN
			n_OutErrId:=112;
		ELSIF bPlatniFent = FALSE THEN
			n_OutErrId:=81;
		END_IF
	20210: // Várakozás a platni elfordulására
		IF (bPlatniBalon = TRUE AND bPlatniJobbon = FALSE) THEN
			IF (s_InCommand='TELJESMERES') THEN
				iState := 800;
			ELSE				
				iState := 20000;
			END_IF
			n_OutErrId := 0;
		ELSIF MAIN.bLevegoOK=FALSE THEN
			n_OutErrId:=5;
		ELSIF bPlatniBalon = FALSE THEN
			n_OutErrId:=107;
		ELSIF bPlatniJobbon = TRUE THEN
			n_OutErrId:=106;
		END_IF

	// Logol
	30000:
		iState := 0;
//		LOGGING.s_InCommand:='LOGOLAS';
	// Leállít
	30001:
		iState := 0;

END_CASE
T_Ticker(IN:= bTickerEnable, PT:= tTickerTime, Q=> bTickerQ, ET=> tTickerET);
TP_hutes(IN:=bHutes, PT:=tHutes, Q=> bAutoHutes, ET=>);
bHutesOn:=(bKeziHutes OR bAutoHutes) AND NOT bHutesTiltas;

CASE iState2 OF
	0:	// Várakozás parancsra
		IF (bStartSchematic=TRUE) THEN
			iState2:=1;
		END_IF
	1:
		IF (bSchematicBusy=TRUE) THEN
			iState2:=2;
		END_IF
	2:
		IF (bSchematicBusy=FALSE) THEN
			bStartSchematic:=FALSE;
			iState2:=0;
		END_IF
END_CASE

// Mérő kapcsolás megnyitása
FB_Start_Schematic(
					NETID:='',
					PATHSTR:='C:\Program Files\Adobe\Reader 11.0\Reader\AcroRd32.exe',
					DIRNAME:='C:\637\',
					COMNDLINE:='"C:\637\590-637-745int-1.pdf"',
					START:=bStartSchematic,
					TMOUT:=T#30S,
					BUSY => bSchematicBusy,
					ERR => bSchematicErr,
					ERRID => nSchematicErr
					);

END_PROGRAM

// ---- POUs/PISTI/Helpers/fb_GetPT1000MinMaxResFromTemp.TcPOU
FUNCTION_BLOCK fb_GetPT1000MinMaxResFromTemp
VAR_INPUT
	rTemp : REAL;
END_VAR
VAR_OUTPUT
	rResMin : REAL := 0;
	rResMax : REAL := 0;
END_VAR
VAR
	rPercent : REAL := 0.01;
END_VAR

rResMin := ((rTemp+259.74)/259.74)*1000*(1-rPercent);
rResMax := ((rTemp+259.74)/259.74)*1000*(1+rPercent);

END_FUNCTION_BLOCK

// ---- POUs/PISTI/Helpers/f_GetPtMinR.TcPOU
FUNCTION f_GetPtMinR : real
VAR_INPUT
	rTemp: REAL := 25;
END_VAR
VAR
	nI: INT;
	rT0, rT1, rR0, rR1, rM: REAL;
END_VAR
VAR CONSTANT
	Pt_MinRT: ARRAY[0..1, 0..15] OF REAL := 
	[0,20,40,60,80,100,120,140,160,180,200,220,240,260,280,300,
	990,1067,1143,1219,1294,1368,1442,1516,1588,1661,1733,1804,1875,1945,2015,2084];
END_VAR

nI:=1;
WHILE (GVL.Pt_NomRT[0,nI]<rTemp) AND (nI<15) DO
	nI:=nI+1;
END_WHILE
rT0:=GVL.Pt_NomRT[0,nI-1];
rT1:=GVL.Pt_NomRT[0,nI];
rR0:=GVL.Pt_NomRT[1,nI-1];
rR1:=GVL.Pt_NomRT[1,nI];
rM:=(rR1-rR0)/(rT1-rT0);
f_GetPtMinR:=(rR0+rM*(rTemp-rT0))/(1+GVL.rPtDev/100);

END_FUNCTION

// ---- POUs/PISTI/Helpers/f_GetPtMaxR.TcPOU
FUNCTION f_GetPtMaxR : real
VAR_INPUT
	rTemp: REAL;
END_VAR
VAR
	nI: INT;
	rT0, rT1, rR0, rR1, rM: REAL;
END_VAR
VAR CONSTANT
	Pt_MaxRT: ARRAY[0..1, 0..15] OF REAL := 
	[0,20,40,60,80,100,120,140,160,180,200,220,240,260,280,300,
	1010,1089,1168,1246,1324,1402,1479,1556,1633,1709,1784,1860,1935,2009,2083,2157];
END_VAR

(*nI:=1;
WHILE (Pt_MaxRT[0,nI]<rTemp) AND (nI<15) DO
	nI:=nI+1;
END_WHILE
rT0:=Pt_MaxRT[0,nI-1];
rT1:=Pt_MaxRT[0,nI];
rR0:=Pt_MaxRT[1,nI-1];
rR1:=Pt_MaxRT[1,nI];
rM:=(rR1-rR0)/(rT1-rT0);
f_GetPtMaxR:=rR0+rM*(rTemp-rT0);*)
nI:=1;
WHILE (GVL.Pt_NomRT[0,nI]<rTemp) AND (nI<15) DO
	nI:=nI+1;
END_WHILE
rT0:=GVL.Pt_NomRT[0,nI-1];
rT1:=GVL.Pt_NomRT[0,nI];
rR0:=GVL.Pt_NomRT[1,nI-1];
rR1:=GVL.Pt_NomRT[1,nI];
rM:=(rR1-rR0)/(rT1-rT0);
f_GetPtMaxR:=(rR0+rM*(rTemp-rT0))*(1+GVL.rPtDev/100);

END_FUNCTION

// ---- POUs/PISTI/Helpers/f_GetNTCMinR.TcPOU
FUNCTION f_GetNTCMinR : real
VAR_INPUT
	rTemp: REAL;
	nProd: UINT;
	rNTCDev: REAL;
END_VAR
VAR
	nI: INT;
	rT0, rT1, rR0, rR1, rM: REAL;
END_VAR
VAR CONSTANT
	rCorr: REAL := 1.1;
	NTC_Sensing_MinRT: ARRAY[0..1, 0..25] OF REAL := 
	[15, 16, 17, 18, 19, 20, 21, 22, 23, 24, 25, 26, 27, 28, 29, 30, 31, 32, 33, 34, 35, 36, 37, 38, 39, 40,
	14966.9, 14299.6, 13665.8, 13063.7, 12491.4, 11947.3, 11430, 10937.9, 10469.8, 10024.2, 9600, 9188.1, 8796.1, 8423, 8067.6, 7729.2, 7406.8, 7099.6, 6806.7, 6527.5, 6261.3, 6007.2, 5764.9, 5533.6, 5312.7, 5101.9];
	NTC_GE_MinRT: ARRAY[0..1, 0..23] OF REAL := 
	[15, 16, 17, 18, 19, 20, 21, 22, 23, 24, 25, 26, 27, 28, 29, 30, 31, 32, 33, 34, 35, 36, 38, 40,
	15133, 14457, 13815, 13206, 12626, 12075, 11552, 11053, 10579, 10128, 9700, 9279.9, 8883.4, 8506.1, 8146.8, 7804.7, 7478.7, 7168.1, 6872.1, 6589.9, 6320.7, 6064, 5585.4, 5149.3];
END_VAR

nI:=1;
(*IF nProd=0 THEN
	WHILE (NTC_Sensing_MinRT[0,nI]<rTemp) AND (nI<25) DO
		nI:=nI+1;
	END_WHILE
	rT0:=NTC_Sensing_MinRT[0,nI-1];
	rT1:=NTC_Sensing_MinRT[0,nI];
	rR0:=NTC_Sensing_MinRT[1,nI-1];
	rR1:=NTC_Sensing_MinRT[1,nI];
	rM:=(rR1-rR0)/(rT1-rT0);
	f_GetNTCMinR:=rR0+rM*(rTemp-rT0);
ELSE
	WHILE (NTC_GE_MinRT[0,nI]<rTemp) AND (nI<23) DO
		nI:=nI+1;
	END_WHILE
	rT0:=NTC_GE_MinRT[0,nI-1];
	rT1:=NTC_GE_MinRT[0,nI];
	rR0:=NTC_GE_MinRT[1,nI-1];
	rR1:=NTC_GE_MinRT[1,nI];
	rM:=(rR1-rR0)/(rT1-rT0);
	f_GetNTCMinR:=rR0+rM*(rTemp-rT0);	
END_IF*)
WHILE (GVL.NTC_Sensing_NomRT[0,nI]<rTemp) AND (nI<25) DO
	nI:=nI+1;
END_WHILE
rT0:=GVL.NTC_Sensing_NomRT[0,nI-1];
rT1:=GVL.NTC_Sensing_NomRT[0,nI];
rR0:=GVL.NTC_Sensing_NomRT[1,nI-1];
rR1:=GVL.NTC_Sensing_NomRT[1,nI];
rM:=(rR1-rR0)/(rT1-rT0);
// f_GetNTCMinR:=(rR0+rM*(rTemp-rT0))/(1+GVL.rNTCDev/100);
f_GetNTCMinR:=(rR0+rM*(rTemp-rT0))/(1+rNTCDev/100);

END_FUNCTION

// ---- POUs/PISTI/Helpers/f_GetNTCMaxR.TcPOU
FUNCTION f_GetNTCMaxR : real
VAR_INPUT
	rTemp: REAL;
	nProd: UINT;
	rNTCDev: REAL;
END_VAR
VAR
	nI: INT;
	rT0, rT1, rR0, rR1, rM: REAL;
END_VAR
VAR CONSTANT
	rCorr: REAL := 1.1;
	NTC_Sensing_MaxRT: ARRAY[0..1, 0..25] OF REAL := 
	[15, 16, 17, 18, 19, 20, 21, 22, 23, 24, 25, 26, 27, 28, 29, 30, 31, 32, 33, 34, 35, 36, 37, 38, 39, 40,
	16360.3, 15616.5, 14910.6, 14240.7, 13604.6, 13000.3, 12426.2, 11880.7, 11362.1, 10869, 10400, 9962.4, 9545.6, 9148.5, 8770.1, 8409.4, 8065.4, 7737.3, 7424.4, 7125.7, 6840.7, 6568.5, 6308.7, 6060.4, 5823.3, 5596.6];
	NTC_GE_MaxRT: ARRAY[0..1, 0..23] OF REAL := 
	[15, 16, 17, 18, 19, 20, 21, 22, 23, 24, 25, 26, 27, 28, 29, 30, 31, 32, 33, 34, 35, 36, 38, 40,
	16214, 15476, 14776, 14111, 13480, 12880, 12311, 11770, 11255, 10766, 10300, 9868.9, 9454.9, 9060.5, 8684.8, 8326.6, 7985.2, 7659.7, 7349.1, 7052.8, 6770.1, 6500.2, 5996.4, 5536.7];
END_VAR

nI:=1;
(*IF nProd=0 THEN
	WHILE (rCorr*GVL.NTC_Sensing_NomRT[0,nI]<rTemp) AND (nI<25) DO
		nI:=nI+1;
	END_WHILE
	rT0:=NTC_Sensing_MaxRT[0,nI-1];
	rT1:=NTC_Sensing_MaxRT[0,nI];
	rR0:=NTC_Sensing_MaxRT[1,nI-1];
	rR1:=NTC_Sensing_MaxRT[1,nI];
	rM:=(rR1-rR0)/(rT1-rT0);
	f_GetNTCMaxR:=rR0+rM*(rTemp-rT0);
ELSE
	WHILE (NTC_GE_MaxRT[0,nI]<rTemp) AND (nI<23) DO
		nI:=nI+1;
	END_WHILE
	rT0:=NTC_GE_MaxRT[0,nI-1];
	rT1:=NTC_GE_MaxRT[0,nI];
	rR0:=NTC_GE_MaxRT[1,nI-1];
	rR1:=NTC_GE_MaxRT[1,nI];
	rM:=(rR1-rR0)/(rT1-rT0);
	f_GetNTCMaxR:=rR0+rM*(rTemp-rT0);
END_IF*)
WHILE (GVL.NTC_Sensing_NomRT[0,nI]<rTemp) AND (nI<25) DO
	nI:=nI+1;
END_WHILE
rT0:=GVL.NTC_Sensing_NomRT[0,nI-1];
rT1:=GVL.NTC_Sensing_NomRT[0,nI];
rR0:=GVL.NTC_Sensing_NomRT[1,nI-1];
rR1:=GVL.NTC_Sensing_NomRT[1,nI];
rM:=(rR1-rR0)/(rT1-rT0);
// f_GetNTCMaxR:=(1+GVL.rNTCDev/100)*(rR0+rM*(rTemp-rT0));
f_GetNTCMaxR:=(1+rNTCDev/100)*(rR0+rM*(rTemp-rT0));

END_FUNCTION

// ---- POUs/PISTI/Helpers/f_GetNTCMinTempFromRes.TcPOU
FUNCTION f_GetNTCMinTempFromRes : REAL
VAR_INPUT
	rRes : REAL;
END_VAR
VAR
	rTemp : REAL := 0;
	rTempTemp : REAL := 0;
END_VAR

IF rRes<>0 THEN 
	rTempTemp := rRes/1000;
	rTempTemp := LN(rTempTemp);
	f_GetNTCMinTempFromRes := rTempTemp*rTempTemp*rTempTemp*(-0.1522);
	f_GetNTCMinTempFromRes := f_GetNTCMinTempFromRes + rTempTemp*rTempTemp*(2.7581);
	f_GetNTCMinTempFromRes := f_GetNTCMinTempFromRes - rTempTemp*(33.077);
	f_GetNTCMinTempFromRes := f_GetNTCMinTempFromRes + 89.119;
ELSE
	f_GetNTCMinTempFromRes := 0;
END_IF

END_FUNCTION

// ---- POUs/PISTI/Helpers/f_GetNTCMaxTempFromRes.TcPOU
FUNCTION f_GetNTCMaxTempFromRes : REAL
VAR_INPUT
	rRes : REAL;
END_VAR
VAR
	rTemp : REAL := 0;
	rTempTemp :REAL := 0;
END_VAR

IF rRes<>0 THEN 
	rTempTemp := rRes/1000;
	rTempTemp := LN(rTempTemp);
	f_GetNTCMaxTempFromRes := rTempTemp*rTempTemp*rTempTemp*(-0.1505);
	f_GetNTCMaxTempFromRes := f_GetNTCMaxTempFromRes + rTempTemp*rTempTemp*(2.563);
	f_GetNTCMaxTempFromRes := f_GetNTCMaxTempFromRes - rTempTemp*(31.865);
	f_GetNTCMaxTempFromRes := f_GetNTCMaxTempFromRes + 85.783;
ELSE
	f_GetNTCMaxTempFromRes := 0;
END_IF

END_FUNCTION

// ---- POUs/PISTI/Helpers/f_GetNTCNomTempFromRes.TcPOU
FUNCTION f_GetNTCNomTempFromRes : REAL
VAR_INPUT
	rRes : REAL;
END_VAR
VAR
	rTemp : REAL := 0;
	rTempTemp :REAL := 0;
END_VAR

IF rRes<>0 THEN 
	rTempTemp := rRes/1000;
	rTempTemp := LN(rTempTemp);
	f_GetNTCNomTempFromRes := rTempTemp*rTempTemp*rTempTemp*(-0.1513);
	f_GetNTCNomTempFromRes := f_GetNTCNomTempFromRes + rTempTemp*rTempTemp*(2.6446);
	f_GetNTCNomTempFromRes := f_GetNTCNomTempFromRes - rTempTemp*(32.485);
	f_GetNTCNomTempFromRes := f_GetNTCNomTempFromRes + 87.472;
ELSE
	f_GetNTCNomTempFromRes := 0;
END_IF

END_FUNCTION

// ---- POUs/PISTI/Helpers/f_GetPTTEMPFromRES.TcPOU
FUNCTION f_GetPTTEMPFromRES : REAL
VAR_INPUT
	rRES : REAL;
END_VAR
VAR
END_VAR

f_GetPTTEMPFromRES := (rRES/1000)*259.74-259.74;

END_FUNCTION

// ---- POUs/GENERAL/Components/HEGESZTOK.TcPOU
PROGRAM HEGESZTOK
VAR
	sHegesztokCommand: STRING := '';
	bHegesztoVorwarnung AT %I*: BOOL;
	bHegesztoElektrodenAnfordem AT %I*: BOOL;
	bHegesztoBereit AT %I*: BOOL;
	bHegesztoStromFehler AT %I*: BOOL;
	bHegesztoMitStromIn AT %I*: BOOL;
	bHegesztoNichtBereit AT %I*: BOOL;
	bHegesztoFK AT %I*: BOOL;
	bHegesztoProgramValasztoOutput AT %Q*:ARRAY [0..4] OF BOOL;
	bHegesztoFejekOutput AT %Q*:ARRAY [0..3] OF BOOL;
	bHegesztoValtoOutput AT %Q*:ARRAY [0..2] OF BOOL;
//	bHegesztoMeldung AT %Q*: BOOL := FALSE;
	bHegeszto3 AT %Q*: BOOL := FALSE;
	iState: INT;
	nHegesztoNumElozo: UINT := 1;
END_VAR
VAR_INPUT
	bHegesztoStart AT %Q*: BOOL := FALSE;		
	nHegesztoNum : UINT := 0;
	bHegesztoMitStromOut AT %Q*: BOOL := FALSE;
END_VAR
VAR_OUTPUT
	ulHegeszto1Utmero AT %I*: ULINT;
	ulHegeszto2Utmero AT %I*: ULINT;
	nError: INT;	
END_VAR
(*VAR_IN_OUT
END_VAR*)

CASE iState OF
	0:	// Új hegesztő programra vár
		IF nHegesztoNum<>nHegesztoNumElozo
			OR (MAIN.bLevegoOK=FALSE AND NOT (nError=0))
			OR (MAIN.bLevegoOK=TRUE AND (nError=1)) THEN
			iState:=1;
		END_IF
		IF bHegesztoStromFehler=TRUE THEN
			nError:=2; // Áramhiba
		END_IF
	1:	// Levegőnyomás ellenőrzése
		IF MAIN.bLevegoOK=TRUE THEN
			nError:=0; // Hibakód törlése
			iState:=2;
		ELSE // B00000=0
			bHegesztoProgramValasztoOutput[0]:=FALSE;
			bHegesztoProgramValasztoOutput[1]:=FALSE;
			bHegesztoProgramValasztoOutput[2]:=FALSE;
			bHegesztoProgramValasztoOutput[3]:=FALSE;
			bHegesztoProgramValasztoOutput[4]:=FALSE;
			bHegesztoFejekOutput[0]:=FALSE;
			bHegesztoFejekOutput[1]:=FALSE;
			bHegesztoFejekOutput[2]:=FALSE;
			bHegesztoFejekOutput[3]:=FALSE;
			bHegesztoValtoOutput[0]:=FALSE;
			bHegesztoValtoOutput[1]:=FALSE;
			bHegesztoValtoOutput[2]:=FALSE;
			bHegeszto3 := FALSE;
			nError:=1; // Nincs levegő
//			iState:=0;
		END_IF
	2:
		CASE nHegesztoNum OF
		//Semelyik
		0:
			bHegesztoProgramValasztoOutput[0]:=TRUE;
			bHegesztoProgramValasztoOutput[1]:=FALSE;
			bHegesztoProgramValasztoOutput[2]:=FALSE;
			bHegesztoProgramValasztoOutput[3]:=FALSE;
			bHegesztoProgramValasztoOutput[4]:=FALSE;
			bHegesztoFejekOutput[0]:=FALSE;
			bHegesztoFejekOutput[1]:=FALSE;
			bHegesztoFejekOutput[2]:=FALSE;
			bHegesztoFejekOutput[3]:=FALSE;
			bHegesztoValtoOutput[0]:=FALSE;
			bHegesztoValtoOutput[1]:=FALSE;
			bHegesztoValtoOutput[2]:=FALSE;
			bHegeszto3 := FALSE;
		//Első fej
		1:	// B00010=2
			bHegesztoProgramValasztoOutput[0]:=FALSE;
			bHegesztoProgramValasztoOutput[1]:=TRUE;
			bHegesztoProgramValasztoOutput[2]:=FALSE;
			bHegesztoProgramValasztoOutput[3]:=FALSE;
			bHegesztoProgramValasztoOutput[4]:=FALSE;
			bHegesztoFejekOutput[0]:=TRUE;
			bHegesztoFejekOutput[1]:=FALSE;
			bHegesztoFejekOutput[2]:=FALSE;
			bHegesztoFejekOutput[3]:=FALSE;
			bHegesztoValtoOutput[0]:=TRUE;
			bHegesztoValtoOutput[1]:=FALSE;
			bHegesztoValtoOutput[2]:=FALSE;
			bHegeszto3 := FALSE;
		2:	// B00011=3
			bHegesztoProgramValasztoOutput[0]:=TRUE;
			bHegesztoProgramValasztoOutput[1]:=TRUE;
			bHegesztoProgramValasztoOutput[2]:=FALSE;
			bHegesztoProgramValasztoOutput[3]:=FALSE;
			bHegesztoProgramValasztoOutput[4]:=FALSE;
			bHegesztoFejekOutput[0]:=TRUE;
			bHegesztoFejekOutput[1]:=FALSE;
			bHegesztoFejekOutput[2]:=FALSE;
			bHegesztoFejekOutput[3]:=FALSE;
			bHegesztoValtoOutput[0]:=TRUE;
			bHegesztoValtoOutput[1]:=FALSE;
			bHegesztoValtoOutput[2]:=FALSE;
			bHegeszto3 := FALSE;
		3:	// B00100=4
			bHegesztoProgramValasztoOutput[0]:=FALSE;
			bHegesztoProgramValasztoOutput[1]:=FALSE;
			bHegesztoProgramValasztoOutput[2]:=TRUE;
			bHegesztoProgramValasztoOutput[3]:=FALSE;
			bHegesztoProgramValasztoOutput[4]:=FALSE;
			bHegesztoFejekOutput[0]:=TRUE;
			bHegesztoFejekOutput[1]:=FALSE;
			bHegesztoFejekOutput[2]:=FALSE;
			bHegesztoFejekOutput[3]:=FALSE;
			bHegesztoValtoOutput[0]:=TRUE;
			bHegesztoValtoOutput[1]:=FALSE;
			bHegesztoValtoOutput[2]:=FALSE;
			bHegeszto3 := FALSE;
		10:	// B01011=11
			bHegesztoProgramValasztoOutput[0]:=TRUE;
			bHegesztoProgramValasztoOutput[1]:=TRUE;
			bHegesztoProgramValasztoOutput[2]:=FALSE;
			bHegesztoProgramValasztoOutput[3]:=TRUE;
			bHegesztoProgramValasztoOutput[4]:=FALSE;
			bHegesztoFejekOutput[0]:=TRUE;
			bHegesztoFejekOutput[1]:=FALSE;
			bHegesztoFejekOutput[2]:=FALSE;
			bHegesztoFejekOutput[3]:=FALSE;
			bHegesztoValtoOutput[0]:=TRUE;
			bHegesztoValtoOutput[1]:=FALSE;
			bHegesztoValtoOutput[2]:=FALSE;
			bHegeszto3 := FALSE;
		11:	// B01100=12
			bHegesztoProgramValasztoOutput[0]:=FALSE;
			bHegesztoProgramValasztoOutput[1]:=FALSE;
			bHegesztoProgramValasztoOutput[2]:=TRUE;
			bHegesztoProgramValasztoOutput[3]:=TRUE;
			bHegesztoProgramValasztoOutput[4]:=FALSE;
			bHegesztoFejekOutput[0]:=TRUE;
			bHegesztoFejekOutput[1]:=FALSE;
			bHegesztoFejekOutput[2]:=FALSE;
			bHegesztoFejekOutput[3]:=FALSE;
			bHegesztoValtoOutput[0]:=TRUE;
			bHegesztoValtoOutput[1]:=FALSE;
			bHegesztoValtoOutput[2]:=FALSE;
			bHegeszto3 := FALSE;
		12:	// B01101=13
			bHegesztoProgramValasztoOutput[0]:=TRUE;
			bHegesztoProgramValasztoOutput[1]:=FALSE;
			bHegesztoProgramValasztoOutput[2]:=TRUE;
			bHegesztoProgramValasztoOutput[3]:=TRUE;
			bHegesztoProgramValasztoOutput[4]:=FALSE;
			bHegesztoFejekOutput[0]:=TRUE;
			bHegesztoFejekOutput[1]:=FALSE;
			bHegesztoFejekOutput[2]:=FALSE;
			bHegesztoFejekOutput[3]:=FALSE;
			bHegesztoValtoOutput[0]:=TRUE;
			bHegesztoValtoOutput[1]:=FALSE;
			bHegesztoValtoOutput[2]:=FALSE;
			bHegeszto3 := FALSE;
		13:	// B01110=14
			bHegesztoProgramValasztoOutput[0]:=FALSE;
			bHegesztoProgramValasztoOutput[1]:=TRUE;
			bHegesztoProgramValasztoOutput[2]:=TRUE;
			bHegesztoProgramValasztoOutput[3]:=TRUE;
			bHegesztoProgramValasztoOutput[4]:=FALSE;
			bHegesztoFejekOutput[0]:=TRUE;
			bHegesztoFejekOutput[1]:=FALSE;
			bHegesztoFejekOutput[2]:=FALSE;
			bHegesztoFejekOutput[3]:=FALSE;
			bHegesztoValtoOutput[0]:=TRUE;
			bHegesztoValtoOutput[1]:=FALSE;
			bHegesztoValtoOutput[2]:=FALSE;
			bHegeszto3 := FALSE;
		//Második fej
		4:	// B00101=5
			bHegesztoProgramValasztoOutput[0]:=TRUE;
			bHegesztoProgramValasztoOutput[1]:=FALSE;
			bHegesztoProgramValasztoOutput[2]:=TRUE;
			bHegesztoProgramValasztoOutput[3]:=FALSE;
			bHegesztoProgramValasztoOutput[4]:=FALSE;
			bHegesztoFejekOutput[0]:=FALSE;
			bHegesztoFejekOutput[1]:=TRUE;
			bHegesztoFejekOutput[2]:=FALSE;
			bHegesztoFejekOutput[3]:=FALSE;
			bHegesztoValtoOutput[0]:=FALSE;
			bHegesztoValtoOutput[1]:=TRUE;
			bHegesztoValtoOutput[2]:=FALSE;
			bHegeszto3 := FALSE;
		5:	// B00110=6
			bHegesztoProgramValasztoOutput[0]:=FALSE;
			bHegesztoProgramValasztoOutput[1]:=TRUE;
			bHegesztoProgramValasztoOutput[2]:=TRUE;
			bHegesztoProgramValasztoOutput[3]:=FALSE;
			bHegesztoProgramValasztoOutput[4]:=FALSE;
			bHegesztoFejekOutput[0]:=FALSE;
			bHegesztoFejekOutput[1]:=TRUE;
			bHegesztoFejekOutput[2]:=FALSE;
			bHegesztoFejekOutput[3]:=FALSE;
			bHegesztoValtoOutput[0]:=FALSE;
			bHegesztoValtoOutput[1]:=TRUE;
			bHegesztoValtoOutput[2]:=FALSE;
			bHegeszto3 := FALSE;
		8:	// B01001=9
			bHegesztoProgramValasztoOutput[0]:=FALSE;
			bHegesztoProgramValasztoOutput[1]:=TRUE;
			bHegesztoProgramValasztoOutput[2]:=FALSE;
			bHegesztoProgramValasztoOutput[3]:=TRUE;
			bHegesztoProgramValasztoOutput[4]:=FALSE;
			bHegesztoFejekOutput[0]:=FALSE;
			bHegesztoFejekOutput[1]:=TRUE;
			bHegesztoFejekOutput[2]:=FALSE;
			bHegesztoFejekOutput[3]:=FALSE;
			bHegesztoValtoOutput[0]:=FALSE;
			bHegesztoValtoOutput[1]:=TRUE;
			bHegesztoValtoOutput[2]:=FALSE;
			bHegeszto3 := FALSE;
		9:	// B01010=10
			bHegesztoProgramValasztoOutput[0]:=FALSE;
			bHegesztoProgramValasztoOutput[1]:=TRUE;
			bHegesztoProgramValasztoOutput[2]:=TRUE;
			bHegesztoProgramValasztoOutput[3]:=FALSE;
			bHegesztoProgramValasztoOutput[4]:=FALSE;
			bHegesztoFejekOutput[0]:=FALSE;
			bHegesztoFejekOutput[1]:=TRUE;
			bHegesztoFejekOutput[2]:=FALSE;
			bHegesztoFejekOutput[3]:=FALSE;
			bHegesztoValtoOutput[0]:=FALSE;
			bHegesztoValtoOutput[1]:=TRUE;
			bHegesztoValtoOutput[2]:=FALSE;
			bHegeszto3 := FALSE;
		//Harmadik fej
		6:	// B00111=7
			bHegesztoProgramValasztoOutput[0]:=TRUE;
			bHegesztoProgramValasztoOutput[1]:=TRUE;
			bHegesztoProgramValasztoOutput[2]:=TRUE;
			bHegesztoProgramValasztoOutput[3]:=FALSE;
			bHegesztoProgramValasztoOutput[4]:=FALSE;
			bHegesztoFejekOutput[0]:=FALSE;
			bHegesztoFejekOutput[1]:=FALSE;
			bHegesztoFejekOutput[2]:=TRUE;
			bHegesztoFejekOutput[3]:=FALSE;
			bHegesztoValtoOutput[0]:=FALSE;
			bHegesztoValtoOutput[1]:=FALSE;
			bHegesztoValtoOutput[2]:=TRUE;
			bHegeszto3 := TRUE;
		7:	// B01000=8
			bHegesztoProgramValasztoOutput[0]:=FALSE;
			bHegesztoProgramValasztoOutput[1]:=FALSE;
			bHegesztoProgramValasztoOutput[2]:=FALSE;
			bHegesztoProgramValasztoOutput[3]:=TRUE;
			bHegesztoProgramValasztoOutput[4]:=FALSE;
			bHegesztoFejekOutput[0]:=FALSE;
			bHegesztoFejekOutput[1]:=FALSE;
			bHegesztoFejekOutput[2]:=TRUE;
			bHegesztoFejekOutput[3]:=FALSE;
			bHegesztoValtoOutput[0]:=FALSE;
			bHegesztoValtoOutput[1]:=FALSE;
			bHegesztoValtoOutput[2]:=TRUE;
			bHegeszto3 := TRUE;
		ELSE // Nem létező program
			bHegesztoProgramValasztoOutput[0]:=FALSE;
			bHegesztoProgramValasztoOutput[1]:=FALSE;
			bHegesztoProgramValasztoOutput[2]:=FALSE;
			bHegesztoProgramValasztoOutput[3]:=FALSE;
			bHegesztoProgramValasztoOutput[4]:=FALSE;
			bHegesztoFejekOutput[0]:=FALSE;
			bHegesztoFejekOutput[1]:=FALSE;
			bHegesztoFejekOutput[2]:=FALSE;
			bHegesztoFejekOutput[3]:=FALSE;
			bHegesztoValtoOutput[0]:=FALSE;
			bHegesztoValtoOutput[1]:=FALSE;
			bHegesztoValtoOutput[2]:=FALSE;
			bHegeszto3 := FALSE;
		END_CASE	
		nHegesztoNumElozo:=nHegesztoNum;
		nError:=100; // Minden rendben
		iState:=0;
END_CASE

// Biztonság
// Ha le kell mennie a hegesztő fejnek, és nincs még lent és benyúltak,
// akkor menjen fel a hegesztő fej
IF ((nHegesztoNum=6) OR (nHegesztoNum=7)) AND (GVL.bHegeszto3Lent=FALSE) THEN
	bHegeszto3:=GVL.bFenysorompoPt;
END_IF

END_PROGRAM

// ---- POUs/PISTI/Components/KAMERAREMOTE.TcPOU
PROGRAM KAMERAREMOTE
VAR
	KameraSocketClose: FB_SocketClose;
	KameraSocketOpen: FB_SocketConnect;
	KameraSocketReceive: FB_SocketReceive;
	KameraSocketSend: FB_SocketSend;
	baReceivedByteArray: ARRAY[0..265] OF BYTE;
	baSendByteArray: ARRAY[0..9] OF BYTE;
	bCloseBusy: BOOL;
	bCloseError: BOOL;
	bConnectBusy: BOOL;
	bConnectError: BOOL;
	bDelayTimePassed: BOOL;
	bReceiveBusy: BOOL;
	bReceiveError: BOOL;
	index: INT;
	bKameraCommOpen : BOOL := FALSE;
	bKameraSocketCloseEnable: BOOL := FALSE;
	bKameraSocketOpenEnable: BOOL := FALSE;
	bKameraSocketReceiveEnable: BOOL := FALSE;
	bKameraSocketSendEnable: BOOL := FALSE;
	bSendBusy: BOOL;
	bSendError: BOOL;
	bStartDelay: BOOL := FALSE;
	Delay: TON;
	hKameraSocket: T_HSOCKET;
	iOpenTrials: INT;
	nCloseErrId: UDINT;
	nConnectErrId: UDINT;
	nReceiveErrId: UDINT;
	nKameraReceivedBytesNum: UDINT;
	nSendErrId: UDINT;
	sKameraRemoteHost: STRING := '192.168.2.40';
	tDelay: TIME;
	uSendByteLen: UDINT := 0;	
	iErrorID: UINT;
	iState2: INT;
	bStartChecker: BOOL;
	FB_Start_Checker: NT_StartProcess;
	bCheckerBusy: BOOL;
	bCheckerErr: BOOL;
	nCheckerErr: UDINT;
END_VAR
VAR_INPUT
	bKameraSetOffline: BOOL;
END_VAR

VAR_OUTPUT
	//Kamera output
	bKameraTriggerReady: BOOL;
	bKameraTriggerAck: BOOL;
	bKameraAcquiring: BOOL;
	bKameraSetup: BOOL;
	bKameraOnline: BOOL;
	bKameraInspecting: BOOL;
	bKameraInspectToggle: BOOL;
	bKameraResultsAvble: BOOL;
	bKameraJobLoaded: BOOL;
	bKameraGeneralFault: BOOL;
	bKameraPartDetect: BOOL;
	bKameraAllPass: BOOL;
	bKameraAnyFail: BOOL;
	bKameraOut00: BOOL;
	bKameraOut01: BOOL;
	bKameraOut02: BOOL;
	bKameraOut03: BOOL;
	bKameraOut04: BOOL;
	bKameraOut05: BOOL;
	bKameraOut06: BOOL;
	bKameraOut07: BOOL;
	
	bIsError : BOOL;
	iState: INT := 0;
END_VAR

VAR_INPUT
	bKameraTrigger: BOOL;
	bKameraTriggerEN: BOOL;
	bKameraCommandSend : BOOL := FALSE;
	bKameraCommOpenEnable : BOOL := FALSE;
	bKameraCommCloseEnable: BOOL := FALSE;
END_VAR

KameraSocketOpen(
			sSrvNetId:= '', 
			sRemoteHost:= sKameraRemoteHost, 
			nRemotePort:= 7733, 
			bExecute:= bKameraSocketOpenEnable, 
			tTimeout:= T#45S, 
			bBusy=> bConnectBusy, 
			bError=> bConnectError, 
			nErrId=> nConnectErrId, 
			hSocket=> hKameraSocket);
			
KameraSocketSend(
			sSrvNetId:= '', 
			hSocket:= hKameraSocket, 
			cbLen:= uSendByteLen, 
			pSrc:= ADR(baSendByteArray), 
			bExecute:= bKameraSocketSendEnable, 
			tTimeout:= T#5S, 
			bBusy=> bSendBusy, 
			bError=> bSendError, 
			nErrId=> nSendErrId);
		
KameraSocketReceive(
			sSrvNetId:= '', 
			hSocket:= hKameraSocket, 
			cbLen:= 266,
			pDest:= ADR(baReceivedByteArray), 
			bExecute:= bKameraSocketReceiveEnable, 
			tTimeout:= T#5S, 
			bBusy=> bReceiveBusy, 
			bError=> bReceiveError, 
			nErrId=> nReceiveErrId, 
			nRecBytes=> nKameraReceivedBytesNum);		
		
KameraSocketClose(
			sSrvNetId:= '', 
			hSocket:= hKameraSocket, 
			bExecute:= bKameraSocketCloseEnable, 
			tTimeout:= T#5S, 
			bBusy=> bCloseBusy, 
			bError=> bCloseError, 
			nErrId=> nCloseErrId);
			
//Kommunikáció nyitás
IF (bKameraCommOpenEnable = TRUE) AND (bKameraCommOpen = FALSE) AND (iState <= 0) THEN
	iState:=1;
	iOpenTrials:=0;
	bIsError:=FALSE;
END_IF;

//Parancs küldés
IF (bKameraCommandSend = TRUE) AND (bKameraCommOpen=TRUE) AND(iState <= 0) THEN
	iState:=11;
	bIsError:=FALSE;
END_IF;

//Kommunikáció zárás
IF (bKameraCommCloseEnable = TRUE) AND (bKameraCommOpen = TRUE) AND (iState <= 0) THEN
	iState:=31;
	bIsError:=FALSE;
END_IF;

//Parancs összeállítás

baSendByteArray[0]:=16#AE;
baSendByteArray[1]:=16#01;

//IF bKameraTriggerEN = TRUE AND bKameraTrigger = FALSE AND bKameraSetOffline = FALSE THEN
//	baSendByteArray[2]:=1;
//ELSIF bKameraTriggerEN = TRUE AND bKameraTrigger =TRUE AND bKameraSetOffline = FALSE THEN
//	baSendByteArray[2]:=3;
//ELSIF bKameraSetOffline = TRUE THEN
//	baSendByteArray[2]:=baSendByteArray[2] OR 128;
//ELSE
//	baSendByteArray[2]:=0;
//END_IF

baSendByteArray[2].0:=bKameraTriggerEN;
baSendByteArray[2].1:=bKameraTrigger;
baSendByteArray[2].7:=bKameraSetOffline;

FOR index:=3 TO 9 DO
	baSendByteArray[index]:=0;
END_FOR


CASE iState OF
	
	1:	//Kommunikáció nyitás
		bKameraSocketOpenEnable:=TRUE;
		iState:=2;
	
	2:
		IF bConnectBusy = TRUE THEN
			iState:=3;
		END_IF
		
	3:
		IF bConnectBusy = FALSE THEN
			iState:=4;
		END_IF 
		
	4:
		IF bConnectError =FALSE THEN
			//Minden OK
			bKameraCommOpen:=TRUE;
			bIsError:=FALSE;
			iState:=0;
		ELSE
			//HIBA
			iOpenTrials:=iOpenTrials+1;
			bKameraCommOpen:=FALSE;
			IF iOpenTrials<6 THEN
				bConnectError:=FALSE;
				iState:=5;
				bStartDelay:=TRUE;
				tDelay:=T#3S;
			ELSE
				iOpenTrials:=0;
				bStartDelay:=FALSE;
				bIsError:=TRUE;
				iErrorID:=340;
				iState:=0;
			END_IF
		END_IF
		bKameraCommOpenEnable := FALSE;
		bKameraSocketOpenEnable:=FALSE;
		
	5:
		IF bDelayTimePassed=TRUE THEN
			bStartDelay:=FALSE;
			iState:=1;
		END_IF

	11: //Parancs küldés
		uSendByteLen := 10;//INT_TO_UDINT(LEN(baSendByteArray));
		//MEMSET(ADR(baReceivedByteArray), 0, 265);
		iState:=12;
		
	12:
		bKameraSocketSendEnable:=TRUE;
		iState:=13;
		
	13:
		IF bSendBusy = TRUE THEN
			iState:=14;
		END_IF
		
	14:
		IF bSendBusy = FALSE THEN
			iState:=15;
		END_IF
		
	15:
		IF bSendError =FALSE THEN
			//Minden OK
			bIsError:= FALSE;
			iState:=21;
		ELSE
			//HIBA
			bIsError:=TRUE;
			iErrorID:=341;
			iState:=0;
		END_IF
		bKameraCommandSend:=FALSE;
		bKameraSocketSendEnable:=FALSE;

	21:	//Adatfogadás
		//nKameraReceivedBytesNum:=0;
		bKameraSocketReceiveEnable:=TRUE;
		iState:=22;
		
	22:
		IF bReceiveBusy = TRUE THEN
			iState:=23;
		END_IF
		
	23:
		IF bReceiveBusy = FALSE THEN
			iState:=24;
		END_IF 
		
	24:
		IF bReceiveError =FALSE THEN
			//Minden OK
			bIsError:= FALSE;
			iState:=25;
		ELSE
			//HIBA
			bIsError:= TRUE;
			iErrorID:=342;
			iState:=0;	
		END_IF
		bKameraSocketReceiveEnable:=FALSE;
		
	25:
		IF (nKameraReceivedBytesNum <> 0) THEN
			iState:=0;
		ELSE
			bIsError:= TRUE;
			iErrorID:=347;
			iState:=0;
		END_IF
		
	31:	//Kommunikáció zárás
		bKameraSocketCloseEnable:=TRUE;
		iState:=32;
		
	32:
		IF bCloseBusy = TRUE THEN
			iState:=33;
		END_IF
		
	33:
		IF bCloseBusy = FALSE THEN
			iState:=34;
		END_IF
		
	34:
		IF bCloseError =FALSE THEN
			//Minden OK
			bIsError:=FALSE;
			bKameraCommOpen:=FALSE;
		ELSE
			//HIBA
			bIsError:=TRUE;
			iErrorID:=343;
			bKameraCommOpen:=FALSE;	//még át kell gondolni
		END_IF
		bKameraCommCloseEnable := FALSE;
		bKameraSocketCloseEnable:=FALSE;
		iState:=0;
	
END_CASE

IF bIsError = FALSE THEN
	iErrorID:=0;
END_IF

//Eredmény kiértékelés

bKameraTriggerReady:=(baReceivedByteArray[0] AND 1)=1;
bKameraTriggerAck:=(baReceivedByteArray[0] AND 2)=2;
bKameraAcquiring:=(baReceivedByteArray[0] AND 4)=4;
bKameraSetup:=(baReceivedByteArray[0] AND 16)=16;
bKameraOnline:=(baReceivedByteArray[0] AND 128)=128;

bKameraInspecting:=(baReceivedByteArray[1] AND 1)=1;
bKameraInspectToggle:=(baReceivedByteArray[1] AND 2)=2;
bKameraResultsAvble:=(baReceivedByteArray[1] AND 8)=8;
bKameraJobLoaded:=(baReceivedByteArray[1] AND 32)=32;
bKameraGeneralFault:=(baReceivedByteArray[1] AND 128)=128;

bKameraPartDetect:=(baReceivedByteArray[2] AND 1)=1;
bKameraAllPass:=(baReceivedByteArray[2] AND 2)=2;
bKameraAnyFail:=(baReceivedByteArray[2] AND 4)=4;

bKameraOut00:=(baReceivedByteArray[3] AND 1)=1;
bKameraOut01:=(baReceivedByteArray[3] AND 2)=2;
bKameraOut02:=(baReceivedByteArray[3] AND 4)=4;
bKameraOut03:=(baReceivedByteArray[3] AND 8)=8;
bKameraOut04:=(baReceivedByteArray[3] AND 16)=16;
bKameraOut05:=(baReceivedByteArray[3] AND 32)=32;
bKameraOut06:=(baReceivedByteArray[3] AND 64)=64;
bKameraOut07:=(baReceivedByteArray[3] AND 128)=128;

Delay(IN:=bStartDelay, PT:=tDelay, Q=>bDelayTimePassed, ET=>);

CASE iState2 OF
	0:	// Várakozás parancsra
		IF (bStartChecker=TRUE) THEN
			iState2:=1;
		END_IF
	1:
		IF (bCheckerBusy=TRUE) THEN
			iState2:=2;
		END_IF
	2:
		IF (bCheckerBusy=FALSE) THEN
			bStartChecker:=FALSE;
			iState2:=0;
		END_IF
END_CASE

// Kamera saját szoftverének indítása
FB_Start_Checker(
					NETID:='',
					PATHSTR:='C:\Program Files\Cognex\Checker Vision Sensors 4.1\Checker.exe',
					DIRNAME:='C:\Program Files\Cognex\Checker Vision Sensors 4.1\',
					COMNDLINE:='',
					START:=bStartChecker,
					TMOUT:=T#30S,
					BUSY => bCheckerBusy,
					ERR => bCheckerErr,
					ERRID => nCheckerErr
					);

END_PROGRAM

// ---- POUs/PISTI/Components/KameraProcess.TcPOU
PROGRAM KameraProcess

VAR
	iState : UDINT := 0;
	b_WaitEnable : BOOL := FALSE;
	b_WaitTime : TIME := T#25MS;
	b_WaitQ : BOOL;
	T_Ticker : TON;
	n_OutErrId: UINT := 0;
END_VAR
VAR_INPUT
	bKameraRun: BOOL;
END_VAR
VAR
	iState2: INT;
	iPartDetectTrials: INT;
	iNotFoundTrials: INT;
	bKameraInspectToggle_Prev: BOOL;
	T_Ticker_2: TON;
	b_WaitEnable_2: BOOL;
	b_WaitTime_2: TIME := T#5s;
	b_WaitQ_2: BOOL;
END_VAR

IF bKameraRun=TRUE THEN
	IF (iState=0 OR iState=1) (*AND n_OutErrId=0*) THEN
		b_WaitEnable:=TRUE;
		iState:=1;
		n_OutErrId:=0;
	END_IF
ELSIF bKameraRun=FALSE AND (iState=0 OR iState=1) THEN
	b_WaitEnable:=FALSE;
END_IF

//IF b_WaitQ=TRUE THEN
	CASE iState OF
		1:	// Kommunikáció kezdeményezése
			IF KAMERAREMOTE.bKameraCommOpen = FALSE THEN
				KAMERAREMOTE.bKameraCommOpenEnable:=TRUE;
			END_IF
			iState := 2;
		2:	// Ha létrejött a kommunikáció
			IF (KAMERAREMOTE.iState = 0) THEN
				IF KAMERAREMOTE.bKameraCommOpen = TRUE AND KAMERAREMOTE.bIsError = FALSE THEN
					iState := 3;
				ELSE
					n_OutErrId:=KAMERAREMOTE.iErrorID;
					iState := 7;
				END_IF;
			END_IF
		3:	// Parancs küldés
			KAMERAREMOTE.bKameraCommandSend := TRUE;
			iState := 4;
		4:	// Ha sikerült a küldés
			IF (KAMERAREMOTE.iState=0) THEN
				IF KAMERAREMOTE.bIsError = FALSE THEN
					iState := 7;
				ELSE
					n_OutErrId := KAMERAREMOTE.iErrorID;
					iState := 7;
				END_IF
			END_IF;
//		5:	// Online állapot ellenőrzése
//			IF KAMERAREMOTE.bKameraOnline = TRUE THEN
//				iState := 7;
//			ELSE
//				n_OutErrId := 344;
//				iState := 7;
//			END_IF
//		6:	//  Trigger Ready ellenőrzése
//			IF KAMERAREMOTE.bKameraTriggerReady = TRUE THEN
//				iState := 7;			
//			ELSE
//				n_OutErrId := 345;
//				iState := 7;
//			END_IF
		7:	// Kommunikáció lezárása
			KAMERAREMOTE.bKameraCommCloseEnable:=TRUE;
			iState := 8;
		8:	// Ha sikerült...
			IF (KAMERAREMOTE.iState=0) THEN
				IF KAMERAREMOTE.bKameraCommOpen = FALSE AND KAMERAREMOTE.bIsError = FALSE THEN
					IF bKameraRun=TRUE THEN
						iState := 9;
					ELSE
						iState := 0;
					END_IF;
				ELSE
					n_OutErrId := KAMERAREMOTE.iErrorID;
					iState := 0;
				END_IF;
			END_IF;
		9:	// Következő tick
			IF b_WaitQ THEN
				iState := 1;
				b_WaitEnable := FALSE;
			END_IF
	END_CASE
//END_IF

T_Ticker(IN:= b_WaitEnable, PT:= b_WaitTime, Q=> b_WaitQ, ET=> );
T_Ticker_2(IN:= b_WaitEnable_2, PT:= b_WaitTime_2, Q=> b_WaitQ_2, ET=> );
//IF b_WaitQ = TRUE THEN
//	b_WaitEnable := FALSE;
//END_IF

IF AUTOMATA.bKameraTrig=TRUE AND bKameraRun=TRUE AND iState2=0 AND n_OutErrId=0 AND GVL.bPtKameraBe=TRUE THEN
	iState2:=1;
ELSIF GVL.bPtKameraBe=FALSE THEN
	iState2:=0;
END_IF

IF NOT b_WaitQ_2 THEN
	CASE iState2 OF
		1:
			AUTOMATA.bKameraTrig:=FALSE;
			iPartDetectTrials:=0;
			iNotFoundTrials:=0;
			b_WaitEnable_2:=TRUE;
			iState2:=2;
		2:
			bKameraInspectToggle_Prev:=KAMERAREMOTE.bKameraInspectToggle;
			KAMERAREMOTE.bKameraTrigger:=TRUE;
			IF KAMERAREMOTE.bKameraTriggerAck=TRUE THEN
				iState2:=4;
				KAMERAREMOTE.bKameraTrigger:=FALSE;
			END_IF
			
		4:
			IF bKameraInspectToggle_Prev<>KAMERAREMOTE.bKameraInspectToggle THEN
				iState2:=5;
			END_IF
		5:
			IF KAMERAREMOTE.bKameraPartDetect=TRUE THEN
				iState2:=6;
			ELSE
				iPartDetectTrials:=iPartDetectTrials+1;
				IF iPartDetectTrials<3 THEN
					iState2:=100;
				ELSE
					n_OutErrId := 344;
					iState2:=0;
				END_IF
			END_IF
		6:
			IF KAMERAREMOTE.bKameraOut04=TRUE OR KAMERAREMOTE.bKameraOut05=TRUE THEN
				iState2:=7;
			ELSE
				iNotFoundTrials:=iNotFoundTrials+1;
				IF iNotFoundTrials<4 THEN
					iState2:=100;
				ELSE
					n_OutErrId := 345;
					iState2:=0;
				END_IF
			END_IF
		7:
			IF KAMERAREMOTE.bKameraTriggerReady=TRUE THEN
				bKameraRun:=FALSE;
				iState2:=0;
			END_IF
		
		
		100: //Ha nem talált Part-ot a kamera, vagy talált, de adaptert vagy kappét nem, újrapróbáljuk 10-szer, csak utána lesz hiba
			IF KAMERAREMOTE.bKameraTriggerReady=TRUE THEN
				iState2:=2;
			END_IF
	END_CASE
ELSE
	iState2:=0;
	b_WaitEnable_2:=FALSE;
	KameraProcess.n_OutErrId:=348;
END_IF

IF n_OutErrId<>0 THEN
	bKameraRun:=FALSE;
	b_WaitEnable:=FALSE;
	b_WaitEnable_2:=FALSE;
	KAMERAREMOTE.bKameraTrigger:=FALSE;
	AUTOMATA.bKameraTrig:=FALSE;
END_IF

END_PROGRAM

// ---- POUs/AUTOMATA.TcPOU
PROGRAM AUTOMATA
VAR	
	iStateElozo: INT := 0;
	iState2Elozo: INT := 0;
	iState: INT := 0;
	iState2: INT := 0;
	bFelfuggeszt: BOOL;
	bFelfuggeszt2: BOOL;
	iCount: INT := 0;
	iCount2: INT := 0;
	bContinue: BOOL := FALSE;
	bContinue2: BOOL := FALSE;
	bContinue2En: BOOL := FALSE;
	bEtalonOK: BOOL := FALSE;
	bRobotReservedBy1: BOOL := FALSE;
	bWelderReservedBy1: BOOL :=FALSE;
	bRobotReservedBy2: BOOL := FALSE;
	bWelderReservedBy2: BOOL :=FALSE;
	bElszivasBe: BOOL := FALSE;
	WAIT: TON;
	WAIT2: TON;
	bStartWait: BOOL := FALSE;
	tWaitTime: TIME;
	bIdoLejart: BOOL := FALSE;
	bStartWait2: BOOL := FALSE;
	tWaitTime2: TIME;
	bIdoLejart2: BOOL := FALSE;
	bHajlitasBe: BOOL := TRUE;
	bHegesztes1Be: BOOL := TRUE;
	bHegesztes2Be: BOOL := TRUE;
	bHegesztes3Be: BOOL := TRUE;
	bHegesztes4Be: BOOL := TRUE;
	bHegesztes5Be: BOOL := TRUE;
	bHegesztes6Be: BOOL := TRUE;
	bHegesztes7Be: BOOL := TRUE;
	bPtKameraBe: BOOL := FALSE;
	bRobotKappeBe: BOOL := TRUE;
	bKappeBe: BOOL := TRUE;
	bMeresBe: BOOL := TRUE;
	bJelolesBe: BOOL := TRUE;
	bUjrameres: BOOL := FALSE;
	bFolyamatBeallitas1Tiltva: BOOL := FALSE;
	bFolyamatBeallitas2Tiltva: BOOL := FALSE;
	bStart1GombNyomva: BOOL := FALSE;
	bStart2GombNyomva: BOOL := FALSE;
	bStart1GombTiltva: BOOL := FALSE;
	bStart2GombTiltva: BOOL := FALSE;
	bPtKameraHasznalatlan: BOOL := FALSE;
	bStopMegnyomva: BOOL;
	sStart1GombFelirat: STRING := 'START';	
	sStop1GombFelirat: STRING := 'Szervízboxhoz';
	sStart2GombFelirat: STRING := 'START';	
	sStop2GombFelirat: STRING := 'Szervízboxhoz';
	sRobotHiba: T_MaxString;
	sExpectedCode: T_MaxString;

	rNTCDev: REAL;
	rPtDev: REAL;
	
	iProductTypeUnderTest: INT;
	
	WATCHDOG: TON;
	bStartWatchDog: BOOL := FALSE;
	tTimeOut: TIME := T#2S;
	bTimeOut: BOOL;
	bWatchDogOK: BOOL;
	
	WATCHDOG2: TON;
	bStartWatchDog2: BOOL := FALSE;
	tTimeOut2: TIME := T#2S;
	bTimeOut2: BOOL;
	bWatchDogOK2: BOOL;
	
	TIMER2: TON;
	bStartTimer2: BOOL := FALSE;
	tTimerTimeOut2: TIME := T#100MS;
	bTimerTimeOut2: BOOL;
	
